// TwinCAT 3 PLC project BE_BUZ_Neutal
// ProgramVersion: 3.1.4023.0
// libraries:
//   EfficientIO Communicator, * (EfficientIO)
//   Lynus Persistent Data V1, * (Lynus AG)
//   Lynus Standards, * (Lynus AG)
//   Tc2_Standard, * (Beckhoff Automation GmbH)
//   Tc2_System, * (Beckhoff Automation GmbH)
//   Tc2_TcpIp, * (Beckhoff Automation GmbH)
//   Tc2_Utilities, * (Beckhoff Automation GmbH)
//   Tc3_IotBase, * (Beckhoff Automation GmbH)
//   Tc3_JsonXml, * (Beckhoff Automation GmbH)
//   Tc3_Module, * (Beckhoff Automation GmbH)
// project tree:
//   / FastTask.TcTTO, MiddleTask.TcTTO, SlowTask.TcTTO
//   FB/ fb_Convert4BytesToLreal.TcPOU, FB_OCHSNER_Web2Com1.TcPOU, FB_OCHSNER_Web2Com2.TcPOU, FB_OCHSNER_Web2Com2_Helper.TcPOU, FB_OCHSNER_Web2Com3_Helper.TcPOU, FB_OCHSNER_Web2Com3.TcPOU, FB_OCHSNER_Web2Com1_Helper.TcPOU, FB_OCHSNER_Web2Com4.TcPOU, FB_OCHSNER_Web2Com4_Helper.TcPOU, FB_TCPModbusRequest_Grid.TcPOU, FB_TCPModbusRequest_PV.TcPOU
//   POUs/ prgComEffIO.TcPOU, prgGrid.TcPOU, prgHP1.TcPOU, prgHP2.TcPOU, prgHP3.TcPOU, prgHP4.TcPOU, prgPersistent.TcPOU, prgPV.TcPOU, prgRWEffIO.TcPOU, prgVarEffIO.TcPOU
// real-time tasks:
//   TASK MiddleTask: cycle T#10ms, priority 8, ADS port 350
//   TASK FastTask: cycle T#5ms, priority 6, ADS port 351
//   TASK SlowTask: cycle T#20ms, priority 10, ADS port 352

CONFIGURATION BE_BUZ_Neutal
    RESOURCE PLC ON TwinCAT3
        TASK FastTask(INTERVAL := T#5ms, PRIORITY := 6);
        TASK MiddleTask(INTERVAL := T#10ms, PRIORITY := 8);
        TASK SlowTask(INTERVAL := T#20ms, PRIORITY := 10);
        PROGRAM prgRWEffIO WITH FastTask : prgRWEffIO;
        PROGRAM prgVarEffIO WITH FastTask : prgVarEffIO;
        PROGRAM prgHP1 WITH MiddleTask : prgHP1;
        PROGRAM prgHP3 WITH MiddleTask : prgHP3;
        PROGRAM prgHP2 WITH MiddleTask : prgHP2;
        PROGRAM prgHP4 WITH MiddleTask : prgHP4;
        PROGRAM prgPV WITH MiddleTask : prgPV;
        PROGRAM prgPersistent WITH MiddleTask : prgPersistent;
        PROGRAM prgComEffIO WITH SlowTask : prgComEffIO;
    END_RESOURCE
END_CONFIGURATION

// ---- POUs/prgRWEffIO.TcPOU
PROGRAM prgRWEffIO
VAR
	fbRW1		: FB_ReadWrite_V2;
END_VAR

fbRW1(
	eUploadType:= eSelectDataUploadType.e_Change_Intervall5min, 
	bBusy=> , 
	bError=> , 
	udiErrorCodeOut=> ,
	eErrorReadWrite_Out=> );

END_PROGRAM

// ---- POUs/prgVarEffIO.TcPOU
PROGRAM prgVarEffIO
VAR
	fbVar			: FB_VarInfo;
END_VAR

fbVar(
	bReadInfo:= , 
	eTMCFile:= eSelectTMCFile.eDontUseTMCFile, 
	eSavePositionTMCFile:= eSavePositionOnPLC.ePostionHardDisk, 
	udiCounterFoundVariables=> , 
	bError=> , 
	bBusy=> , 
	byProgress=> , 
	udiErrorCodeOut=> , 
	eErrorVarInfo_Out=> , 
	sVarWithError=> );

END_PROGRAM

// ---- POUs/prgHP1.TcPOU
PROGRAM prgHP1
VAR
	fbWb2Com1						: FB_OCHSNER_Web2Com1;
	byHP1StateHeatProd		: BYTE;		//{#lynus.ag#()}
	lrHP1TWVtemp			: LREAL;	//{#lynus.ag#()}
	lrHP1TWRtemp			: LREAL;	//{#lynus.ag#()}
	lrHP1TQAtemp			: LREAL;	//{#lynus.ag#()}
	lrHP1TQEtemp			: LREAL;	//{#lynus.ag#()}
	lrHP1ThEnergykWh		: LREAL;	//{#lynus.ag#()}
	lrHP1ThEnergyMWh		: LREAL;	//{#lynus.ag#()}
	byHC1StateHC			: BYTE;		//{#lynus.ag#()}
	lrHC1OutTemp			: LREAL;	//{#lynus.ag#()}
	lrHC1OutTempAvg			: LREAL;	//{#lynus.ag#()}
	lrHC1SPRoomTemp			: LREAL;	//{#lynus.ag#()}
	lrHC1PreFlowTemp		: LREAL;	//{#lynus.ag#()}
	lrHC1SPFlowTemp			: LREAL;	//{#lynus.ag#()}
	byHP2StateHeatProd		: BYTE;		//{#lynus.ag#()}
	lrHP2TWVtemp			: LREAL;	//{#lynus.ag#()}
	lrHP2TWRtemp			: LREAL;	//{#lynus.ag#()}
	lrHP2TQAtemp			: LREAL;	//{#lynus.ag#()}
	lrHP2TQEtemp			: LREAL;	//{#lynus.ag#()}
	lrHP2ThEnergykWh		: LREAL;	//{#lynus.ag#()}
	lrHP2ThEnergyMWh		: LREAL;	//{#lynus.ag#()}
END_VAR

fbWb2Com1(
	bStart:= TRUE, 
	tDelayRequest:= T#60S, 
	sHostname:= 'localhost', 
	bValidResult=> , 
	bBusy=> , 
	bError=> , 
	bDone=> , 
	hrErrorCode=> ,
	byHP1StateHeatProd => byHP1StateHeatProd,
	lrHP1TWVtemp => lrHP1TWVtemp,
	lrHP1TWRtemp => lrHP1TWRtemp,
	lrHP1TQAtemp => lrHP1TQAtemp,
	lrHP1TQEtemp => lrHP1TQEtemp,
	lrHP1ThEnergykWh => lrHP1ThEnergykWh,
	lrHP1ThEnergyMWh => lrHP1ThEnergyMWh,
	byHC1StateHC => byHC1StateHC,
	lrHC1OutTemp => lrHC1OutTemp,
	lrHC1OutTempAvg => lrHC1OutTempAvg,
	lrHC1SPRoomTemp => lrHC1SPRoomTemp,
	lrHC1PreFlowTemp => lrHC1PreFlowTemp,
	lrHC1SPFlowTemp => lrHC1SPFlowTemp,
	byHP2StateHeatProd => byHP2StateHeatProd,
	lrHP2TWVtemp => lrHP2TWVtemp,
	lrHP2TWRtemp => lrHP2TWRtemp,
	lrHP2TQAtemp => lrHP2TQAtemp,
	lrHP2TQEtemp => lrHP2TQEtemp,
	lrHP2ThEnergykWh => lrHP2ThEnergykWh,
	lrHP2ThEnergyMWh => lrHP2ThEnergyMWh);

END_PROGRAM

// ---- FB/FB_OCHSNER_Web2Com1.TcPOU
FUNCTION_BLOCK FB_OCHSNER_Web2Com1
VAR_INPUT
	bStart				: BOOL;
	tDelayRequest		: TIME;		//Timer for delay before start with the next read or write Request
	sHostname			: STRING(255);		//Hostname or IP Adress from the Server
END_VAR

VAR_IN_OUT
END_VAR

VAR_OUTPUT
	bValidResult		: BOOL;							//Valid Result received from Server
    bBusy				: BOOL;							//Function is Busy
    bError				: BOOL;							//Error sucess
	bDone				: BOOL;							//True after the decoding from the received Json File
	bConnected			: BOOL;							//Connection to the Server
	hrErrorCode       	: HRESULT;						//Error Result from Http Client
	byHP1StateHeatProd		: BYTE;
	lrHP1TWVtemp			: LREAL;
	lrHP1TWRtemp			: LREAL;
	lrHP1TQAtemp			: LREAL;
	lrHP1TQEtemp			: LREAL;
	lrHP1ThEnergykWh		: LREAL;
	lrHP1ThEnergyMWh		: LREAL;
	byHC1StateHC			: BYTE;
	lrHC1OutTemp			: LREAL;
	lrHC1OutTempAvg			: LREAL;
	lrHC1SPRoomTemp			: LREAL;
	lrHC1PreFlowTemp		: LREAL;
	lrHC1SPFlowTemp			: LREAL;
	byHP2StateHeatProd		: BYTE;
	lrHP2TWVtemp			: LREAL;
	lrHP2TWRtemp			: LREAL;
	lrHP2TQAtemp			: LREAL;
	lrHP2TQEtemp			: LREAL;
	lrHP2ThEnergykWh		: LREAL;
	lrHP2ThEnergyMWh		: LREAL;
END_VAR

VAR
	fbClient			: FB_IotHttpClient;
	fbHttpGet			: FB_OCHSNER_Web2Com1_Helper;
	timStartRequest		: TON;							//Timer to Start the Request
	FPStartRequest		: R_TRIG;						//Internal positive Edge
	FPDone				: R_TRIG;						//Internal positive Edge
	FNStart				: F_TRIG;						//Internal negative Edge
END_VAR

(*------------------------------------------------------------------------------------Configure HTTP Client------------------------------------------------------------------------------------------------------*)

fbClient.sHostName := sHostname;
fbClient.tConnectionTimeout := T#20S;
fbClient.bKeepAlive := FALSE;

IF NOT fbClient.bConfigured THEN 
	fbClient.nHostPort:= 80;
	fbClient.bKeepAlive := FALSE;
	fbClient.tConnectionTimeout := T#20S;
END_IF


//Timer to start the Request
FPStartRequest(CLK:= bStart, Q=> );
	timStartRequest(IN:= fbClient.bConfigured AND bStart AND NOT timStartRequest.Q, PT:= tDelayRequest, Q=> , ET=> );
		IF ((timStartRequest.Q AND NOT bBusy) OR (FPStartRequest.Q AND NOT bBusy AND fbClient.bConfigured)) THEN fbHttpGet.bSend := TRUE; END_IF

				
//Http Get Function
fbHttpGet(
	bSend:= , 
	fbClient:= fbClient, 
	bBusy=> bBusy, 
	bError=> ,
	byHP1StateHeatProd => byHP1StateHeatProd,
	lrHP1TWVtemp => lrHP1TWVtemp,
	lrHP1TWRtemp => lrHP1TWRtemp,
	lrHP1TQAtemp => lrHP1TQAtemp,
	lrHP1TQEtemp => lrHP1TQEtemp,
	lrHP1ThEnergykWh => lrHP1ThEnergykWh,
	lrHP1ThEnergyMWh => lrHP1ThEnergyMWh,
	byHC1StateHC => byHC1StateHC,
	lrHC1OutTemp => lrHC1OutTemp,
	lrHC1OutTempAvg => lrHC1OutTempAvg,
	lrHC1SPRoomTemp => lrHC1SPRoomTemp,
	lrHC1PreFlowTemp => lrHC1PreFlowTemp,
	lrHC1SPFlowTemp => lrHC1SPFlowTemp,
	byHP2StateHeatProd => byHP2StateHeatProd,
	lrHP2TWVtemp => lrHP2TWVtemp,
	lrHP2TWRtemp => lrHP2TWRtemp,
	lrHP2TQAtemp => lrHP2TQAtemp,
	lrHP2TQEtemp => lrHP2TQEtemp,
	lrHP2ThEnergykWh => lrHP2ThEnergykWh,
	lrHP2ThEnergyMWh => lrHP2ThEnergyMWh );


fbHttpGet.bSend := FALSE;

FPDone(CLK:= bDone, Q=> );

fbClient.Execute();

//Error
IF fbHttpGet.bError OR fbClient.bError THEN bError := TRUE; ELSE bError := FALSE; END_IF	
	hrErrorCode := fbClient.hrErrorCode;

END_FUNCTION_BLOCK

// ---- FB/FB_OCHSNER_Web2Com1_Helper.TcPOU
FUNCTION_BLOCK FB_OCHSNER_Web2Com1_Helper
VAR_INPUT
	bSend				: BOOL;
END_VAR

VAR_IN_OUT
	fbClient			: FB_IotHttpClient;
END_VAR

VAR_OUTPUT
	bBusy				: BOOL;
	bError				: BOOL;
	byHP1StateHeatProd		: BYTE;
	lrHP1TWVtemp			: LREAL;
	lrHP1TWRtemp			: LREAL;
	lrHP1TQAtemp			: LREAL;
	lrHP1TQEtemp			: LREAL;
	lrHP1ThEnergykWh		: LREAL;
	lrHP1ThEnergyMWh		: LREAL;
	byHC1StateHC			: BYTE;
	lrHC1OutTemp			: LREAL;
	lrHC1OutTempAvg			: LREAL;
	lrHC1SPRoomTemp			: LREAL;
	lrHC1PreFlowTemp		: LREAL;
	lrHC1SPFlowTemp			: LREAL;
	byHP2StateHeatProd		: BYTE;
	lrHP2TWVtemp			: LREAL;
	lrHP2TWRtemp			: LREAL;
	lrHP2TQAtemp			: LREAL;
	lrHP2TQEtemp			: LREAL;
	lrHP2ThEnergykWh		: LREAL;
	lrHP2ThEnergyMWh		: LREAL;
END_VAR

VAR
	fbRequest1			: FB_IotHttpRequest;
	fbRequest2			: FB_IotHttpRequest;
	fbRequest3			: FB_IotHttpRequest;

	fbJson				: FB_JsonDomParser;
	nState				: UDINT;
	RisingEdge			: R_TRIG;
	timTimeout			: TON;
	tTimeOut			: TIME := T#90S;
	bGetContentResult	: BOOL;
	sContent1			: STRING(511);
	sContent2			: STRING(511);
	sContent3			: STRING(511);
	
	bGetJsonResult		: BOOL;
	jsonDoc				: SJsonValue;
	jsonVal				: SJsonValue;
	
	nReqCount			: UDINT;	
	nResCount			: UDINT;
	nValidResCount		: UDINT;
	nErrCount			: UDINT;
END_VAR

//Timer for Timeout
timTimeout(IN:= nState = 1 AND bBusy, PT:= tTimeOut, Q=> , ET=> );
	IF timTimeout.Q THEN 
		nState := 0;
		bBusy := FALSE;
	END_IF

RisingEdge(CLK:= bSend );
CASE nState OF
0:	
	IF RisingEdge.Q THEN 
		IF 
			fbRequest1.SendRequest(sUri:='/web2com_1HP1.php', fbClient:=fbClient, eRequestType:=ETcIotHttpRequestType.HTTP_Get, 0, 0, 0) AND
			fbRequest2.SendRequest(sUri:='/web2com_1HC1.php', fbClient:=fbClient, eRequestType:=ETcIotHttpRequestType.HTTP_Get, 0, 0, 0) AND 
			fbRequest3.SendRequest(sUri:='/web2com_1HP2.php', fbClient:=fbClient, eRequestType:=ETcIotHttpRequestType.HTTP_Get, 0, 0, 0) THEN				
			nState:= 1;
			nReqCount:= nReqCount+1;
			bBusy:= TRUE;
			bError:= FALSE;
		END_IF					
	END_IF
1:
	IF NOT fbRequest1.bBusy AND NOT fbRequest2.bBusy AND NOT fbRequest3.bBusy THEN
		bError:= TRUE;
		IF NOT fbRequest1.bError THEN				 
			bGetContentResult:= fbRequest1.GetContent(pContent:= ADR(sContent1), nContentSize:= SIZEOF(sContent1), bSetNullTermination:= TRUE);
			IF fbRequest1.nStatusCode >= 200 AND fbRequest1.nStatusCode < 300 THEN
				bGetJsonResult:= FALSE;
				jsonDoc:= fbRequest1.GetJsonDomContent(fbJson);
				IF jsonDoc <> 0 THEN
					bGetJsonResult:= TRUE;
					IF fbJson.HasMember(jsonDoc, '1211250')  THEN
						jsonVal:= fbJson.FindMember(jsonDoc, '1211250');
						nValidResCount:= nValidResCount+1;
						IF fbJson.IsNumber(jsonVal) THEN							
							byHP1StateHeatProd := DINT_TO_BYTE(fbJson.GetInt(jsonVal));									
						END_IF
						
						jsonVal:= fbJson.FindMember(jsonDoc, '1211251');
						nValidResCount:= nValidResCount+1;
						IF fbJson.IsDouble(jsonVal) THEN							
							lrHP1TWVtemp := fbJson.GetDouble(jsonVal);									
						END_IF
						
						jsonVal:= fbJson.FindMember(jsonDoc, '1211253');
						nValidResCount:= nValidResCount+1;
						IF fbJson.IsDouble(jsonVal) THEN							
							lrHP1TWRtemp := fbJson.GetDouble(jsonVal);									
						END_IF
						
						jsonVal:= fbJson.FindMember(jsonDoc, '1211254');
						nValidResCount:= nValidResCount+1;
						IF fbJson.IsDouble(jsonVal) THEN							
							lrHP1TQAtemp := fbJson.GetDouble(jsonVal);									
						END_IF
						
						jsonVal:= fbJson.FindMember(jsonDoc, '1211255');
						nValidResCount:= nValidResCount+1;
						IF fbJson.IsDouble(jsonVal) THEN							
							lrHP1TQEtemp := fbJson.GetDouble(jsonVal);									
						END_IF
						
						jsonVal:= fbJson.FindMember(jsonDoc, '1211258');
						nValidResCount:= nValidResCount+1;
						IF fbJson.IsNumber(jsonVal) THEN							
							lrHP1ThEnergykWh := fbJson.GetDouble(jsonVal);									
						END_IF
						
						jsonVal:= fbJson.FindMember(jsonDoc, '1211259');
						nValidResCount:= nValidResCount+1;
						IF fbJson.IsNumber(jsonVal) THEN							
							lrHP1ThEnergyMWh := fbJson.GetDouble(jsonVal);									
						END_IF
						
						bError:= FALSE;
						END_IF
					END_IF						
				nResCount:= nResCount+1;			
				END_IF
		END_IF
		
		IF NOT fbRequest2.bError THEN				 
			bGetContentResult:= fbRequest2.GetContent(pContent:= ADR(sContent2), nContentSize:= SIZEOF(sContent2), bSetNullTermination:= TRUE);
			IF fbRequest2.nStatusCode >= 200 AND fbRequest2.nStatusCode < 300 THEN
				bGetJsonResult:= FALSE;
				jsonDoc:= fbRequest2.GetJsonDomContent(fbJson);
				IF jsonDoc <> 0 THEN
					bGetJsonResult:= TRUE;
					IF fbJson.HasMember(jsonDoc, '1241190')  THEN
						jsonVal:= fbJson.FindMember(jsonDoc, '1241190');
						nValidResCount:= nValidResCount+1;
						IF fbJson.IsNumber(jsonVal) THEN							
							byHC1StateHC := DINT_TO_BYTE(fbJson.GetInt(jsonVal));									
						END_IF
						
						jsonVal:= fbJson.FindMember(jsonDoc, '1241191');
						nValidResCount:= nValidResCount+1;
						IF fbJson.IsDouble(jsonVal) THEN							
							lrHC1OutTemp := fbJson.GetDouble(jsonVal);									
						END_IF
						
						jsonVal:= fbJson.FindMember(jsonDoc, '1241192');
						nValidResCount:= nValidResCount+1;
						IF fbJson.IsDouble(jsonVal) THEN							
							lrHC1OutTempAvg := fbJson.GetDouble(jsonVal);									
						END_IF
						
						jsonVal:= fbJson.FindMember(jsonDoc, '1241193');
						nValidResCount:= nValidResCount+1;
						IF fbJson.IsDouble(jsonVal) THEN							
							lrHC1SPRoomTemp := fbJson.GetDouble(jsonVal);									
						END_IF
						
						jsonVal:= fbJson.FindMember(jsonDoc, '1241194');
						nValidResCount:= nValidResCount+1;
						IF fbJson.IsDouble(jsonVal) THEN							
							lrHC1PreFlowTemp := fbJson.GetDouble(jsonVal);									
						END_IF
						
						jsonVal:= fbJson.FindMember(jsonDoc, '1241195');
						nValidResCount:= nValidResCount+1;
						IF fbJson.IsDouble(jsonVal) THEN							
							lrHC1SPFlowTemp := fbJson.GetDouble(jsonVal);									
						END_IF
						
						bError:= FALSE;
						END_IF
					END_IF						
				nResCount:= nResCount+1;			
				END_IF
		END_IF
		
		IF NOT fbRequest3.bError THEN				 
			bGetContentResult:= fbRequest3.GetContent(pContent:= ADR(sContent3), nContentSize:= SIZEOF(sContent3), bSetNullTermination:= TRUE);
			IF fbRequest3.nStatusCode >= 200 AND fbRequest3.nStatusCode < 300 THEN
				bGetJsonResult:= FALSE;
				jsonDoc:= fbRequest3.GetJsonDomContent(fbJson);
				IF jsonDoc <> 0 THEN
					bGetJsonResult:= TRUE;
					IF fbJson.HasMember(jsonDoc, '1311250')  THEN
						jsonVal:= fbJson.FindMember(jsonDoc, '1311250');
						nValidResCount:= nValidResCount+1;
						IF fbJson.IsNumber(jsonVal) THEN							
							byHP2StateHeatProd := DINT_TO_BYTE(fbJson.GetInt(jsonVal));									
						END_IF
						
						jsonVal:= fbJson.FindMember(jsonDoc, '1311251');
						nValidResCount:= nValidResCount+1;
						IF fbJson.IsDouble(jsonVal) THEN							
							lrHP2TWVtemp := fbJson.GetDouble(jsonVal);									
						END_IF
						
						jsonVal:= fbJson.FindMember(jsonDoc, '1311253');
						nValidResCount:= nValidResCount+1;
						IF fbJson.IsDouble(jsonVal) THEN							
							lrHP2TWRtemp := fbJson.GetDouble(jsonVal);									
						END_IF
						
						jsonVal:= fbJson.FindMember(jsonDoc, '1311254');
						nValidResCount:= nValidResCount+1;
						IF fbJson.IsDouble(jsonVal) THEN							
							lrHP2TQAtemp := fbJson.GetDouble(jsonVal);									
						END_IF
						
						jsonVal:= fbJson.FindMember(jsonDoc, '1311255');
						nValidResCount:= nValidResCount+1;
						IF fbJson.IsDouble(jsonVal) THEN							
							lrHP2TQEtemp := fbJson.GetDouble(jsonVal);									
						END_IF
						
						jsonVal:= fbJson.FindMember(jsonDoc, '1311258');
						nValidResCount:= nValidResCount+1;
						IF fbJson.IsNumber(jsonVal) THEN							
							lrHP2ThEnergykWh := fbJson.GetDouble(jsonVal);									
						END_IF
						
						jsonVal:= fbJson.FindMember(jsonDoc, '1311259');
						nValidResCount:= nValidResCount+1;
						IF fbJson.IsNumber(jsonVal) THEN							
							lrHP2ThEnergyMWh := fbJson.GetDouble(jsonVal);									
						END_IF
						
						bError:= FALSE;
						END_IF
					END_IF						
				nResCount:= nResCount+1;			
				END_IF
		END_IF
		
		nState:= 0;
		bBusy:= FALSE;
		IF bError THEN
			nErrCount:= nErrCount+1;
		END_IF
	END_IF  	
END_CASE

END_FUNCTION_BLOCK

// ---- POUs/prgHP3.TcPOU
PROGRAM prgHP3
VAR
	fbWb2Com3						: FB_OCHSNER_Web2Com3;
	byHP1StateHeatProd		: BYTE;		//{#lynus.ag#()}
	lrHP1TWVtemp			: LREAL;	//{#lynus.ag#()}
	lrHP1TWRtemp			: LREAL;	//{#lynus.ag#()}
	lrHP1TQAtemp			: LREAL;	//{#lynus.ag#()}
	lrHP1TQEtemp			: LREAL;	//{#lynus.ag#()}
	lrHP1ThEnergykWh		: LREAL;	//{#lynus.ag#()}
	lrHP1ThEnergyMWh		: LREAL;	//{#lynus.ag#()}
	byHC1StateHC			: BYTE;		//{#lynus.ag#()}
	lrHC1OutTemp			: LREAL;	//{#lynus.ag#()}
	lrHC1OutTempAvg			: LREAL;	//{#lynus.ag#()}
	lrHC1RoomTemp			: LREAL;	//{#lynus.ag#()}
	lrHC1SPRoomTemp			: LREAL;	//{#lynus.ag#()}
	lrHC1PreFlowTemp		: LREAL;	//{#lynus.ag#()}
	lrHC1SPFlowTemp			: LREAL;	//{#lynus.ag#()}
END_VAR

fbWb2Com3(
	bStart:= TRUE, 
	tDelayRequest:= T#60S, 
	sHostname:= 'localhost', 
	bValidResult=> , 
	bBusy=> , 
	bError=> , 
	bDone=> , 
	hrErrorCode=> ,
	byHP1StateHeatProd => byHP1StateHeatProd,
	lrHP1TWVtemp => lrHP1TWVtemp,
	lrHP1TWRtemp => lrHP1TWRtemp,
	lrHP1TQAtemp => lrHP1TQAtemp,
	lrHP1TQEtemp => lrHP1TQEtemp,
	lrHP1ThEnergykWh => lrHP1ThEnergykWh,
	lrHP1ThEnergyMWh => lrHP1ThEnergyMWh,
	byHC1StateHC => byHC1StateHC,
	lrHC1OutTemp => lrHC1OutTemp,
	lrHC1OutTempAvg => lrHC1OutTempAvg,
	lrHC1RoomTemp => lrHC1RoomTemp,
	lrHC1SPRoomTemp => lrHC1SPRoomTemp,
	lrHC1PreFlowTemp => lrHC1PreFlowTemp,
	lrHC1SPFlowTemp => lrHC1SPFlowTemp);

END_PROGRAM

// ---- FB/FB_OCHSNER_Web2Com3.TcPOU
FUNCTION_BLOCK FB_OCHSNER_Web2Com3
VAR_INPUT
	bStart				: BOOL;
	tDelayRequest		: TIME;		//Timer for delay before start with the next read or write Request
	sHostname			: STRING(255);		//Hostname or IP Adress from the Server
END_VAR

VAR_IN_OUT
END_VAR

VAR_OUTPUT
	bValidResult		: BOOL;							//Valid Result received from Server
    bBusy				: BOOL;							//Function is Busy
    bError				: BOOL;							//Error sucess
	bDone				: BOOL;							//True after the decoding from the received Json File
	bConnected			: BOOL;							//Connection to the Server
	hrErrorCode       	: HRESULT;						//Error Result from Http Client
	byHP1StateHeatProd		: BYTE;
	lrHP1TWVtemp			: LREAL;
	lrHP1TWRtemp			: LREAL;
	lrHP1TQAtemp			: LREAL;
	lrHP1TQEtemp			: LREAL;
	lrHP1ThEnergykWh		: LREAL;
	lrHP1ThEnergyMWh		: LREAL;
	byHC1StateHC			: BYTE;
	lrHC1OutTemp			: LREAL;
	lrHC1OutTempAvg			: LREAL;
	lrHC1RoomTemp			: LREAL;
	lrHC1SPRoomTemp			: LREAL;
	lrHC1PreFlowTemp		: LREAL;
	lrHC1SPFlowTemp			: LREAL;
END_VAR

VAR
	fbClient			: FB_IotHttpClient;
	fbHttpGet			: FB_OCHSNER_Web2Com3_Helper;
	timStartRequest		: TON;							//Timer to Start the Request
	FPStartRequest		: R_TRIG;						//Internal positive Edge
	FPDone				: R_TRIG;						//Internal positive Edge
	FNStart				: F_TRIG;						//Internal negative Edge
END_VAR

(*------------------------------------------------------------------------------------Configure HTTP Client------------------------------------------------------------------------------------------------------*)

fbClient.sHostName := sHostname;
fbClient.tConnectionTimeout := T#20S;
fbClient.bKeepAlive := FALSE;

IF NOT fbClient.bConfigured THEN 
	fbClient.nHostPort:= 80;
	fbClient.bKeepAlive := FALSE;
	fbClient.tConnectionTimeout := T#20S;
END_IF


//Timer to start the Request
FPStartRequest(CLK:= bStart, Q=> );
	timStartRequest(IN:= fbClient.bConfigured AND bStart AND NOT timStartRequest.Q, PT:= tDelayRequest, Q=> , ET=> );
		IF ((timStartRequest.Q AND NOT bBusy) OR (FPStartRequest.Q AND NOT bBusy AND fbClient.bConfigured)) THEN fbHttpGet.bSend := TRUE; END_IF

				
//Http Get Function
fbHttpGet(
	bSend:= , 
	fbClient:= fbClient, 
	bBusy=> bBusy, 
	bError=> ,
	byHP1StateHeatProd => byHP1StateHeatProd,
	lrHP1TWVtemp => lrHP1TWVtemp,
	lrHP1TWRtemp => lrHP1TWRtemp,
	lrHP1TQAtemp => lrHP1TQAtemp,
	lrHP1TQEtemp => lrHP1TQEtemp,
	lrHP1ThEnergykWh => lrHP1ThEnergykWh,
	lrHP1ThEnergyMWh => lrHP1ThEnergyMWh,
	byHC1StateHC => byHC1StateHC,
	lrHC1OutTemp => lrHC1OutTemp,
	lrHC1OutTempAvg => lrHC1OutTempAvg,
	lrHC1RoomTemp => lrHC1RoomTemp,
	lrHC1SPRoomTemp => lrHC1SPRoomTemp,
	lrHC1PreFlowTemp => lrHC1PreFlowTemp,
	lrHC1SPFlowTemp => lrHC1SPFlowTemp);


fbHttpGet.bSend := FALSE;

FPDone(CLK:= bDone, Q=> );

fbClient.Execute();

//Error
IF fbHttpGet.bError OR fbClient.bError THEN bError := TRUE; ELSE bError := FALSE; END_IF	
	hrErrorCode := fbClient.hrErrorCode;

END_FUNCTION_BLOCK

// ---- FB/FB_OCHSNER_Web2Com3_Helper.TcPOU
FUNCTION_BLOCK FB_OCHSNER_Web2Com3_Helper
VAR_INPUT
	bSend				: BOOL;
END_VAR

VAR_IN_OUT
	fbClient			: FB_IotHttpClient;
END_VAR

VAR_OUTPUT
	bBusy				: BOOL;
	bError				: BOOL;
	byHP1StateHeatProd		: BYTE;
	lrHP1TWVtemp			: LREAL;
	lrHP1TWRtemp			: LREAL;
	lrHP1TQAtemp			: LREAL;
	lrHP1TQEtemp			: LREAL;
	lrHP1ThEnergykWh		: LREAL;
	lrHP1ThEnergyMWh		: LREAL;
	byHC1StateHC			: BYTE;
	lrHC1OutTemp			: LREAL;
	lrHC1OutTempAvg			: LREAL;
	lrHC1RoomTemp			: LREAL;
	lrHC1SPRoomTemp			: LREAL;
	lrHC1PreFlowTemp		: LREAL;
	lrHC1SPFlowTemp			: LREAL;
END_VAR

VAR
	fbRequest1			: FB_IotHttpRequest;
	fbRequest2			: FB_IotHttpRequest;

	fbJson				: FB_JsonDomParser;
	nState				: UDINT;
	RisingEdge			: R_TRIG;
	timTimeout			: TON;
	tTimeOut			: TIME := T#90S;
	bGetContentResult	: BOOL;
	sContent1			: STRING(511);
	sContent2			: STRING(511);
	
	bGetJsonResult		: BOOL;
	jsonDoc				: SJsonValue;
	jsonVal				: SJsonValue;
	
	nReqCount			: UDINT;	
	nResCount			: UDINT;
	nValidResCount		: UDINT;
	nErrCount			: UDINT;
END_VAR

//Timer for Timeout
timTimeout(IN:= nState = 1 AND bBusy, PT:= tTimeOut, Q=> , ET=> );
	IF timTimeout.Q THEN 
		nState := 0;
		bBusy := FALSE;
	END_IF

RisingEdge(CLK:= bSend );
CASE nState OF
0:	
	IF RisingEdge.Q THEN 
		IF 
			fbRequest1.SendRequest(sUri:='/web2com_3HP1.php', fbClient:=fbClient, eRequestType:=ETcIotHttpRequestType.HTTP_Get, 0, 0, 0) AND
			fbRequest2.SendRequest(sUri:='/web2com_3HC1.php', fbClient:=fbClient, eRequestType:=ETcIotHttpRequestType.HTTP_Get, 0, 0, 0) THEN				
			nState:= 1;
			nReqCount:= nReqCount+1;
			bBusy:= TRUE;
			bError:= FALSE;
		END_IF					
	END_IF
1:
	IF NOT fbRequest1.bBusy AND NOT fbRequest2.bBusy THEN
		bError:= TRUE;
		IF NOT fbRequest1.bError THEN				 
			bGetContentResult:= fbRequest1.GetContent(pContent:= ADR(sContent1), nContentSize:= SIZEOF(sContent1), bSetNullTermination:= TRUE);
			IF fbRequest1.nStatusCode >= 200 AND fbRequest1.nStatusCode < 300 THEN
				bGetJsonResult:= FALSE;
				jsonDoc:= fbRequest1.GetJsonDomContent(fbJson);
				IF jsonDoc <> 0 THEN
					bGetJsonResult:= TRUE;
					IF fbJson.HasMember(jsonDoc, '1211250')  THEN
						jsonVal:= fbJson.FindMember(jsonDoc, '1211250');
						nValidResCount:= nValidResCount+1;
						IF fbJson.IsNumber(jsonVal) THEN							
							byHP1StateHeatProd := DINT_TO_BYTE(fbJson.GetInt(jsonVal));									
						END_IF
						
						jsonVal:= fbJson.FindMember(jsonDoc, '1211251');
						nValidResCount:= nValidResCount+1;
						IF fbJson.IsDouble(jsonVal) THEN							
							lrHP1TWVtemp := fbJson.GetDouble(jsonVal);									
						END_IF
						
						jsonVal:= fbJson.FindMember(jsonDoc, '1211253');
						nValidResCount:= nValidResCount+1;
						IF fbJson.IsDouble(jsonVal) THEN							
							lrHP1TWRtemp := fbJson.GetDouble(jsonVal);									
						END_IF
						
						jsonVal:= fbJson.FindMember(jsonDoc, '1211254');
						nValidResCount:= nValidResCount+1;
						IF fbJson.IsDouble(jsonVal) THEN							
							lrHP1TQAtemp := fbJson.GetDouble(jsonVal);									
						END_IF
						
						jsonVal:= fbJson.FindMember(jsonDoc, '1211255');
						nValidResCount:= nValidResCount+1;
						IF fbJson.IsDouble(jsonVal) THEN							
							lrHP1TQEtemp := fbJson.GetDouble(jsonVal);									
						END_IF
						
						jsonVal:= fbJson.FindMember(jsonDoc, '1211258');
						nValidResCount:= nValidResCount+1;
						IF fbJson.IsNumber(jsonVal) THEN							
							lrHP1ThEnergykWh := fbJson.GetDouble(jsonVal);									
						END_IF
						
						jsonVal:= fbJson.FindMember(jsonDoc, '1211259');
						nValidResCount:= nValidResCount+1;
						IF fbJson.IsNumber(jsonVal) THEN							
							lrHP1ThEnergyMWh := fbJson.GetDouble(jsonVal);									
						END_IF
						
						bError:= FALSE;
						END_IF
					END_IF						
				nResCount:= nResCount+1;			
				END_IF
		END_IF
		
		IF NOT fbRequest2.bError THEN				 
			bGetContentResult:= fbRequest2.GetContent(pContent:= ADR(sContent2), nContentSize:= SIZEOF(sContent2), bSetNullTermination:= TRUE);
			IF fbRequest2.nStatusCode >= 200 AND fbRequest2.nStatusCode < 300 THEN
				bGetJsonResult:= FALSE;
				jsonDoc:= fbRequest2.GetJsonDomContent(fbJson);
				IF jsonDoc <> 0 THEN
					bGetJsonResult:= TRUE;
					IF fbJson.HasMember(jsonDoc, '1241190')  THEN
						jsonVal:= fbJson.FindMember(jsonDoc, '1241190');
						nValidResCount:= nValidResCount+1;
						IF fbJson.IsNumber(jsonVal) THEN							
							byHC1StateHC := DINT_TO_BYTE(fbJson.GetInt(jsonVal));									
						END_IF
						
						jsonVal:= fbJson.FindMember(jsonDoc, '1241191');
						nValidResCount:= nValidResCount+1;
						IF fbJson.IsDouble(jsonVal) THEN							
							lrHC1OutTemp := fbJson.GetDouble(jsonVal);									
						END_IF
						
						jsonVal:= fbJson.FindMember(jsonDoc, '1241192');
						nValidResCount:= nValidResCount+1;
						IF fbJson.IsDouble(jsonVal) THEN							
							lrHC1OutTempAvg := fbJson.GetDouble(jsonVal);									
						END_IF
						
						jsonVal:= fbJson.FindMember(jsonDoc, '1241193');
						nValidResCount:= nValidResCount+1;
						IF fbJson.IsDouble(jsonVal) THEN							
							lrHC1RoomTemp := fbJson.GetDouble(jsonVal);									
						END_IF
						
						jsonVal:= fbJson.FindMember(jsonDoc, '1241194');
						nValidResCount:= nValidResCount+1;
						IF fbJson.IsDouble(jsonVal) THEN							
							lrHC1SPRoomTemp := fbJson.GetDouble(jsonVal);									
						END_IF
						
						jsonVal:= fbJson.FindMember(jsonDoc, '1241195');
						nValidResCount:= nValidResCount+1;
						IF fbJson.IsDouble(jsonVal) THEN							
							lrHC1PreFlowTemp := fbJson.GetDouble(jsonVal);									
						END_IF
						
						jsonVal:= fbJson.FindMember(jsonDoc, '1241196');
						nValidResCount:= nValidResCount+1;
						IF fbJson.IsDouble(jsonVal) THEN							
							lrHC1SPFlowTemp := fbJson.GetDouble(jsonVal);									
						END_IF
						
						bError:= FALSE;
						END_IF
					END_IF						
				nResCount:= nResCount+1;			
				END_IF
		END_IF
		
		nState:= 0;
		bBusy:= FALSE;
		IF bError THEN
			nErrCount:= nErrCount+1;
		END_IF
	END_IF  	
END_CASE

END_FUNCTION_BLOCK

// ---- POUs/prgHP2.TcPOU
PROGRAM prgHP2
VAR
	fbWb2Com2						: FB_OCHSNER_Web2Com2;
	byHP1StateHeatProd		: BYTE;		//{#lynus.ag#()}
	lrHP1TWVtemp			: LREAL;	//{#lynus.ag#()}
	lrHP1TWRtemp			: LREAL;	//{#lynus.ag#()}
	lrHP1TQAtemp			: LREAL;	//{#lynus.ag#()}
	lrHP1TQEtemp			: LREAL;	//{#lynus.ag#()}
	lrHP1ThEnergykWh		: LREAL;	//{#lynus.ag#()}
	lrHP1ThEnergyMWh		: LREAL;	//{#lynus.ag#()}
	byHC1StateHC			: BYTE;
	lrHC1OutTemp			: LREAL;
	lrHC1OutTempAvg			: LREAL;
	lrHC1SPRoomTemp			: LREAL;
	lrHC1PreFlowTemp		: LREAL;
	lrHC1SPFlowTemp			: LREAL;
END_VAR

fbWb2Com2(
	bStart:= TRUE, 
	tDelayRequest:= T#60S, 
	sHostname:= 'localhost', 
	bValidResult=> , 
	bBusy=> , 
	bError=> , 
	bDone=> , 
	hrErrorCode=> ,
	byHP1StateHeatProd => byHP1StateHeatProd,
	lrHP1TWVtemp => lrHP1TWVtemp,
	lrHP1TWRtemp => lrHP1TWRtemp,
	lrHP1TQAtemp => lrHP1TQAtemp,
	lrHP1TQEtemp => lrHP1TQEtemp,
	lrHP1ThEnergykWh => lrHP1ThEnergykWh,
	lrHP1ThEnergyMWh => lrHP1ThEnergyMWh,
	byHC1StateHC => byHC1StateHC,
	lrHC1OutTemp => lrHC1OutTemp,
	lrHC1OutTempAvg => lrHC1OutTempAvg,
	lrHC1SPRoomTemp => lrHC1SPRoomTemp,
	lrHC1PreFlowTemp => lrHC1PreFlowTemp,
	lrHC1SPFlowTemp => lrHC1SPFlowTemp);

END_PROGRAM

// ---- FB/FB_OCHSNER_Web2Com2.TcPOU
FUNCTION_BLOCK FB_OCHSNER_Web2Com2
VAR_INPUT
	bStart				: BOOL;
	tDelayRequest		: TIME;		//Timer for delay before start with the next read or write Request
	sHostname			: STRING(255);		//Hostname or IP Adress from the Server
END_VAR

VAR_IN_OUT
END_VAR

VAR_OUTPUT
	bValidResult		: BOOL;							//Valid Result received from Server
    bBusy				: BOOL;							//Function is Busy
    bError				: BOOL;							//Error sucess
	bDone				: BOOL;							//True after the decoding from the received Json File
	bConnected			: BOOL;							//Connection to the Server
	hrErrorCode       	: HRESULT;						//Error Result from Http Client
	byHP1StateHeatProd		: BYTE;
	lrHP1TWVtemp			: LREAL;
	lrHP1TWRtemp			: LREAL;
	lrHP1TQAtemp			: LREAL;
	lrHP1TQEtemp			: LREAL;
	lrHP1ThEnergykWh		: LREAL;
	lrHP1ThEnergyMWh		: LREAL;
	byHC1StateHC			: BYTE;
	lrHC1OutTemp			: LREAL;
	lrHC1OutTempAvg			: LREAL;
	lrHC1RoomTemp			: LREAL;
	lrHC1SPRoomTemp			: LREAL;
	lrHC1PreFlowTemp		: LREAL;
	lrHC1SPFlowTemp			: LREAL;
END_VAR

VAR
	fbClient			: FB_IotHttpClient;
	fbHttpGet			: FB_OCHSNER_Web2Com2_Helper;
	timStartRequest		: TON;							//Timer to Start the Request
	FPStartRequest		: R_TRIG;						//Internal positive Edge
	FPDone				: R_TRIG;						//Internal positive Edge
	FNStart				: F_TRIG;						//Internal negative Edge
END_VAR

(*------------------------------------------------------------------------------------Configure HTTP Client------------------------------------------------------------------------------------------------------*)

fbClient.sHostName := sHostname;
fbClient.tConnectionTimeout := T#20S;
fbClient.bKeepAlive := FALSE;

IF NOT fbClient.bConfigured THEN 
	fbClient.nHostPort:= 80;
	fbClient.bKeepAlive := FALSE;
	fbClient.tConnectionTimeout := T#20S;
END_IF


//Timer to start the Request
FPStartRequest(CLK:= bStart, Q=> );
	timStartRequest(IN:= fbClient.bConfigured AND bStart AND NOT timStartRequest.Q, PT:= tDelayRequest, Q=> , ET=> );
		IF ((timStartRequest.Q AND NOT bBusy) OR (FPStartRequest.Q AND NOT bBusy AND fbClient.bConfigured)) THEN fbHttpGet.bSend := TRUE; END_IF

				
//Http Get Function
fbHttpGet(
	bSend:= , 
	fbClient:= fbClient, 
	bBusy=> bBusy, 
	bError=> ,
	byHP1StateHeatProd => byHP1StateHeatProd,
	lrHP1TWVtemp => lrHP1TWVtemp,
	lrHP1TWRtemp => lrHP1TWRtemp,
	lrHP1TQAtemp => lrHP1TQAtemp,
	lrHP1TQEtemp => lrHP1TQEtemp,
	lrHP1ThEnergykWh => lrHP1ThEnergykWh,
	lrHP1ThEnergyMWh => lrHP1ThEnergyMWh,
	byHC1StateHC => byHC1StateHC,
	lrHC1OutTemp => lrHC1OutTemp,
	lrHC1OutTempAvg => lrHC1OutTempAvg,
	lrHC1RoomTemp => lrHC1RoomTemp,
	lrHC1SPRoomTemp => lrHC1SPRoomTemp,
	lrHC1PreFlowTemp => lrHC1PreFlowTemp,
	lrHC1SPFlowTemp => lrHC1SPFlowTemp);


fbHttpGet.bSend := FALSE;

FPDone(CLK:= bDone, Q=> );

fbClient.Execute();

//Error
IF fbHttpGet.bError OR fbClient.bError THEN bError := TRUE; ELSE bError := FALSE; END_IF	
	hrErrorCode := fbClient.hrErrorCode;

END_FUNCTION_BLOCK

// ---- FB/FB_OCHSNER_Web2Com2_Helper.TcPOU
FUNCTION_BLOCK FB_OCHSNER_Web2Com2_Helper
VAR_INPUT
	bSend				: BOOL;
END_VAR

VAR_IN_OUT
	fbClient			: FB_IotHttpClient;
END_VAR

VAR_OUTPUT
	bBusy				: BOOL;
	bError				: BOOL;
	byHP1StateHeatProd		: BYTE;
	lrHP1TWVtemp			: LREAL;
	lrHP1TWRtemp			: LREAL;
	lrHP1TQAtemp			: LREAL;
	lrHP1TQEtemp			: LREAL;
	lrHP1ThEnergykWh		: LREAL;
	lrHP1ThEnergyMWh		: LREAL;
	byHC1StateHC			: BYTE;
	lrHC1OutTemp			: LREAL;
	lrHC1OutTempAvg			: LREAL;
	lrHC1RoomTemp			: LREAL;
	lrHC1SPRoomTemp			: LREAL;
	lrHC1PreFlowTemp		: LREAL;
	lrHC1SPFlowTemp			: LREAL;
END_VAR

VAR
	fbRequest1			: FB_IotHttpRequest;
	fbRequest2			: FB_IotHttpRequest;

	fbJson				: FB_JsonDomParser;
	nState				: UDINT;
	RisingEdge			: R_TRIG;
	timTimeout			: TON;
	tTimeOut			: TIME := T#90S;
	bGetContentResult	: BOOL;
	sContent1			: STRING(511);
	sContent2			: STRING(511);
	
	bGetJsonResult		: BOOL;
	jsonDoc				: SJsonValue;
	jsonVal				: SJsonValue;
	
	nReqCount			: UDINT;	
	nResCount			: UDINT;
	nValidResCount		: UDINT;
	nErrCount			: UDINT;
END_VAR

//Timer for Timeout
timTimeout(IN:= nState = 1 AND bBusy, PT:= tTimeOut, Q=> , ET=> );
	IF timTimeout.Q THEN 
		nState := 0;
		bBusy := FALSE;
	END_IF

RisingEdge(CLK:= bSend );
CASE nState OF
0:	
	IF RisingEdge.Q THEN 
		IF 
			fbRequest1.SendRequest(sUri:='/web2com_2HP1.php', fbClient:=fbClient, eRequestType:=ETcIotHttpRequestType.HTTP_Get, 0, 0, 0) THEN				
			nState:= 1;
			nReqCount:= nReqCount+1;
			bBusy:= TRUE;
			bError:= FALSE;
		END_IF					
	END_IF
1:
	IF NOT fbRequest1.bBusy THEN
		bError:= TRUE;
		IF NOT fbRequest1.bError THEN				 
			bGetContentResult:= fbRequest1.GetContent(pContent:= ADR(sContent1), nContentSize:= SIZEOF(sContent1), bSetNullTermination:= TRUE);
			IF fbRequest1.nStatusCode >= 200 AND fbRequest1.nStatusCode < 300 THEN
				bGetJsonResult:= FALSE;
				jsonDoc:= fbRequest1.GetJsonDomContent(fbJson);
				IF jsonDoc <> 0 THEN
					bGetJsonResult:= TRUE;
					IF fbJson.HasMember(jsonDoc, '1211250')  THEN
						jsonVal:= fbJson.FindMember(jsonDoc, '1211250');
						nValidResCount:= nValidResCount+1;
						IF fbJson.IsNumber(jsonVal) THEN							
							byHP1StateHeatProd := DINT_TO_BYTE(fbJson.GetInt(jsonVal));									
						END_IF
						
						jsonVal:= fbJson.FindMember(jsonDoc, '1211251');
						nValidResCount:= nValidResCount+1;
						IF fbJson.IsDouble(jsonVal) THEN							
							lrHP1TWVtemp := fbJson.GetDouble(jsonVal);									
						END_IF
						
						jsonVal:= fbJson.FindMember(jsonDoc, '1211252');
						nValidResCount:= nValidResCount+1;
						IF fbJson.IsDouble(jsonVal) THEN							
							lrHP1TWRtemp := fbJson.GetDouble(jsonVal);									
						END_IF
						
						jsonVal:= fbJson.FindMember(jsonDoc, '1211253');
						nValidResCount:= nValidResCount+1;
						IF fbJson.IsDouble(jsonVal) THEN							
							lrHP1TQAtemp := fbJson.GetDouble(jsonVal);									
						END_IF
						
						jsonVal:= fbJson.FindMember(jsonDoc, '1211254');
						nValidResCount:= nValidResCount+1;
						IF fbJson.IsDouble(jsonVal) THEN							
							lrHP1TQEtemp := fbJson.GetDouble(jsonVal);									
						END_IF
						
						jsonVal:= fbJson.FindMember(jsonDoc, '1211258');
						nValidResCount:= nValidResCount+1;
						IF fbJson.IsNumber(jsonVal) THEN							
							lrHP1ThEnergykWh := fbJson.GetDouble(jsonVal);									
						END_IF
						
						jsonVal:= fbJson.FindMember(jsonDoc, '1211259');
						nValidResCount:= nValidResCount+1;
						IF fbJson.IsNumber(jsonVal) THEN							
							lrHP1ThEnergyMWh := fbJson.GetDouble(jsonVal);									
						END_IF
						
						bError:= FALSE;
						END_IF
					END_IF						
				nResCount:= nResCount+1;			
				END_IF
		END_IF
		(*
		IF NOT fbRequest2.bError THEN				 
			bGetContentResult:= fbRequest2.GetContent(pContent:= ADR(sContent2), nContentSize:= SIZEOF(sContent2), bSetNullTermination:= TRUE);
			IF fbRequest2.nStatusCode >= 200 AND fbRequest2.nStatusCode < 300 THEN
				bGetJsonResult:= FALSE;
				jsonDoc:= fbRequest2.GetJsonDomContent(fbJson);
				IF jsonDoc <> 0 THEN
					bGetJsonResult:= TRUE;
					IF fbJson.HasMember(jsonDoc, '1241190')  THEN
						jsonVal:= fbJson.FindMember(jsonDoc, '1241190');
						nValidResCount:= nValidResCount+1;
						IF fbJson.IsNumber(jsonVal) THEN							
							byHC1StateHC := DINT_TO_BYTE(fbJson.GetInt(jsonVal));									
						END_IF
						
						jsonVal:= fbJson.FindMember(jsonDoc, '1241191');
						nValidResCount:= nValidResCount+1;
						IF fbJson.IsDouble(jsonVal) THEN							
							lrHC1OutTemp := fbJson.GetDouble(jsonVal);									
						END_IF
						
						jsonVal:= fbJson.FindMember(jsonDoc, '1241192');
						nValidResCount:= nValidResCount+1;
						IF fbJson.IsDouble(jsonVal) THEN							
							lrHC1OutTempAvg := fbJson.GetDouble(jsonVal);									
						END_IF
						
						jsonVal:= fbJson.FindMember(jsonDoc, '1241193');
						nValidResCount:= nValidResCount+1;
						IF fbJson.IsDouble(jsonVal) THEN							
							lrHC1RoomTemp := fbJson.GetDouble(jsonVal);									
						END_IF
						
						jsonVal:= fbJson.FindMember(jsonDoc, '1241194');
						nValidResCount:= nValidResCount+1;
						IF fbJson.IsDouble(jsonVal) THEN							
							lrHC1SPRoomTemp := fbJson.GetDouble(jsonVal);									
						END_IF
						
						jsonVal:= fbJson.FindMember(jsonDoc, '1241195');
						nValidResCount:= nValidResCount+1;
						IF fbJson.IsDouble(jsonVal) THEN							
							lrHC1PreFlowTemp := fbJson.GetDouble(jsonVal);									
						END_IF
						
						jsonVal:= fbJson.FindMember(jsonDoc, '1241196');
						nValidResCount:= nValidResCount+1;
						IF fbJson.IsDouble(jsonVal) THEN							
							lrHC1SPFlowTemp := fbJson.GetDouble(jsonVal);									
						END_IF
						
						bError:= FALSE;
						END_IF
					END_IF						
				nResCount:= nResCount+1;			
				END_IF
		END_IF
		*)
		nState:= 0;
		bBusy:= FALSE;
		IF bError THEN
			nErrCount:= nErrCount+1;
		END_IF
	END_IF  	
END_CASE

END_FUNCTION_BLOCK

// ---- POUs/prgHP4.TcPOU
PROGRAM prgHP4
VAR
	fbWb2Com4						: FB_OCHSNER_Web2Com4;
	byHP1StateHeatProd		: BYTE;		//{#lynus.ag#()}
	lrHP1TWVtemp			: LREAL;	//{#lynus.ag#()}
	lrHP1TWRtemp			: LREAL;	//{#lynus.ag#()}
	lrHP1TQAtemp			: LREAL;	//{#lynus.ag#()}
	lrHP1TQEtemp			: LREAL;	//{#lynus.ag#()}
	lrHP1ThEnergykWh		: LREAL;	//{#lynus.ag#()}
	lrHP1ThEnergyMWh		: LREAL;	//{#lynus.ag#()}
	byHC1StateHC			: BYTE;		//{#lynus.ag#()}
	lrHC1OutTemp			: LREAL;	//{#lynus.ag#()}
	lrHC1OutTempAvg			: LREAL;	//{#lynus.ag#()}
	lrHC1SPRoomTemp			: LREAL;	//{#lynus.ag#()}
	lrHC1PreFlowTemp		: LREAL;	//{#lynus.ag#()}
	lrHC1SPFlowTemp			: LREAL;	//{#lynus.ag#()}
END_VAR

fbWb2Com4(
	bStart:= TRUE, 
	tDelayRequest:= T#60S, 
	sHostname:= 'localhost', 
	bValidResult=> , 
	bBusy=> , 
	bError=> , 
	bDone=> , 
	hrErrorCode=> ,
	byHP1StateHeatProd => byHP1StateHeatProd,
	lrHP1TWVtemp => lrHP1TWVtemp,
	lrHP1TWRtemp => lrHP1TWRtemp,
	lrHP1TQAtemp => lrHP1TQAtemp,
	lrHP1TQEtemp => lrHP1TQEtemp,
	lrHP1ThEnergykWh => lrHP1ThEnergykWh,
	lrHP1ThEnergyMWh => lrHP1ThEnergyMWh,
	byHC1StateHC => byHC1StateHC,
	lrHC1OutTemp => lrHC1OutTemp,
	lrHC1OutTempAvg => lrHC1OutTempAvg,
	lrHC1SPRoomTemp => lrHC1SPRoomTemp,
	lrHC1PreFlowTemp => lrHC1PreFlowTemp,
	lrHC1SPFlowTemp => lrHC1SPFlowTemp);

END_PROGRAM

// ---- FB/FB_OCHSNER_Web2Com4.TcPOU
FUNCTION_BLOCK FB_OCHSNER_Web2Com4
VAR_INPUT
	bStart				: BOOL;
	tDelayRequest		: TIME;		//Timer for delay before start with the next read or write Request
	sHostname			: STRING(255);		//Hostname or IP Adress from the Server
END_VAR

VAR_IN_OUT
END_VAR

VAR_OUTPUT
	bValidResult		: BOOL;							//Valid Result received from Server
    bBusy				: BOOL;							//Function is Busy
    bError				: BOOL;							//Error sucess
	bDone				: BOOL;							//True after the decoding from the received Json File
	bConnected			: BOOL;							//Connection to the Server
	hrErrorCode       	: HRESULT;						//Error Result from Http Client
	byHP1StateHeatProd		: BYTE;
	lrHP1TWVtemp			: LREAL;
	lrHP1TWRtemp			: LREAL;
	lrHP1TQAtemp			: LREAL;
	lrHP1TQEtemp			: LREAL;
	lrHP1ThEnergykWh		: LREAL;
	lrHP1ThEnergyMWh		: LREAL;
	byHC1StateHC			: BYTE;
	lrHC1OutTemp			: LREAL;
	lrHC1OutTempAvg			: LREAL;
	lrHC1RoomTemp			: LREAL;
	lrHC1SPRoomTemp			: LREAL;
	lrHC1PreFlowTemp		: LREAL;
	lrHC1SPFlowTemp			: LREAL;
END_VAR

VAR
	fbClient			: FB_IotHttpClient;
	fbHttpGet			: FB_OCHSNER_Web2Com4_Helper;
	timStartRequest		: TON;							//Timer to Start the Request
	FPStartRequest		: R_TRIG;						//Internal positive Edge
	FPDone				: R_TRIG;						//Internal positive Edge
	FNStart				: F_TRIG;						//Internal negative Edge
END_VAR

(*------------------------------------------------------------------------------------Configure HTTP Client------------------------------------------------------------------------------------------------------*)

fbClient.sHostName := sHostname;
fbClient.tConnectionTimeout := T#20S;
fbClient.bKeepAlive := FALSE;

IF NOT fbClient.bConfigured THEN 
	fbClient.nHostPort:= 80;
	fbClient.bKeepAlive := FALSE;
	fbClient.tConnectionTimeout := T#20S;
END_IF


//Timer to start the Request
FPStartRequest(CLK:= bStart, Q=> );
	timStartRequest(IN:= fbClient.bConfigured AND bStart AND NOT timStartRequest.Q, PT:= tDelayRequest, Q=> , ET=> );
		IF ((timStartRequest.Q AND NOT bBusy) OR (FPStartRequest.Q AND NOT bBusy AND fbClient.bConfigured)) THEN fbHttpGet.bSend := TRUE; END_IF

				
//Http Get Function
fbHttpGet(
	bSend:= , 
	fbClient:= fbClient, 
	bBusy=> bBusy, 
	bError=> ,
	byHP1StateHeatProd => byHP1StateHeatProd,
	lrHP1TWVtemp => lrHP1TWVtemp,
	lrHP1TWRtemp => lrHP1TWRtemp,
	lrHP1TQAtemp => lrHP1TQAtemp,
	lrHP1TQEtemp => lrHP1TQEtemp,
	lrHP1ThEnergykWh => lrHP1ThEnergykWh,
	lrHP1ThEnergyMWh => lrHP1ThEnergyMWh,
	byHC1StateHC => byHC1StateHC,
	lrHC1OutTemp => lrHC1OutTemp,
	lrHC1OutTempAvg => lrHC1OutTempAvg,
	lrHC1SPRoomTemp => lrHC1SPRoomTemp,
	lrHC1PreFlowTemp => lrHC1PreFlowTemp,
	lrHC1SPFlowTemp => lrHC1SPFlowTemp);


fbHttpGet.bSend := FALSE;

FPDone(CLK:= bDone, Q=> );

fbClient.Execute();

//Error
IF fbHttpGet.bError OR fbClient.bError THEN bError := TRUE; ELSE bError := FALSE; END_IF	
	hrErrorCode := fbClient.hrErrorCode;

END_FUNCTION_BLOCK

// ---- FB/FB_OCHSNER_Web2Com4_Helper.TcPOU
FUNCTION_BLOCK FB_OCHSNER_Web2Com4_Helper
VAR_INPUT
	bSend				: BOOL;
END_VAR

VAR_IN_OUT
	fbClient			: FB_IotHttpClient;
END_VAR

VAR_OUTPUT
	bBusy				: BOOL;
	bError				: BOOL;
	byHP1StateHeatProd		: BYTE;
	lrHP1TWVtemp			: LREAL;
	lrHP1TWRtemp			: LREAL;
	lrHP1TQAtemp			: LREAL;
	lrHP1TQEtemp			: LREAL;
	lrHP1ThEnergykWh		: LREAL;
	lrHP1ThEnergyMWh		: LREAL;
	byHC1StateHC			: BYTE;
	lrHC1OutTemp			: LREAL;
	lrHC1OutTempAvg			: LREAL;
	lrHC1SPRoomTemp			: LREAL;
	lrHC1PreFlowTemp		: LREAL;
	lrHC1SPFlowTemp			: LREAL;
END_VAR

VAR
	fbRequest1			: FB_IotHttpRequest;
	fbRequest2			: FB_IotHttpRequest;

	fbJson				: FB_JsonDomParser;
	nState				: UDINT;
	RisingEdge			: R_TRIG;
	timTimeout			: TON;
	tTimeOut			: TIME := T#90S;
	bGetContentResult	: BOOL;
	sContent1			: STRING(511);
	sContent2			: STRING(511);
	
	bGetJsonResult		: BOOL;
	jsonDoc				: SJsonValue;
	jsonVal				: SJsonValue;
	
	nReqCount			: UDINT;	
	nResCount			: UDINT;
	nValidResCount		: UDINT;
	nErrCount			: UDINT;
END_VAR

//Timer for Timeout
timTimeout(IN:= nState = 1 AND bBusy, PT:= tTimeOut, Q=> , ET=> );
	IF timTimeout.Q THEN 
		nState := 0;
		bBusy := FALSE;
	END_IF

RisingEdge(CLK:= bSend );
CASE nState OF
0:	
	IF RisingEdge.Q THEN 
		IF 
			fbRequest1.SendRequest(sUri:='/web2com_4HP1.php', fbClient:=fbClient, eRequestType:=ETcIotHttpRequestType.HTTP_Get, 0, 0, 0) AND
			fbRequest2.SendRequest(sUri:='/web2com_4HC1.php', fbClient:=fbClient, eRequestType:=ETcIotHttpRequestType.HTTP_Get, 0, 0, 0) THEN				
			nState:= 1;
			nReqCount:= nReqCount+1;
			bBusy:= TRUE;
			bError:= FALSE;
		END_IF					
	END_IF
1:
	IF NOT fbRequest1.bBusy AND NOT fbRequest2.bBusy THEN
		bError:= TRUE;
		IF NOT fbRequest1.bError THEN				 
			bGetContentResult:= fbRequest1.GetContent(pContent:= ADR(sContent1), nContentSize:= SIZEOF(sContent1), bSetNullTermination:= TRUE);
			IF fbRequest1.nStatusCode >= 200 AND fbRequest1.nStatusCode < 300 THEN
				bGetJsonResult:= FALSE;
				jsonDoc:= fbRequest1.GetJsonDomContent(fbJson);
				IF jsonDoc <> 0 THEN
					bGetJsonResult:= TRUE;
					IF fbJson.HasMember(jsonDoc, '1211250')  THEN
						jsonVal:= fbJson.FindMember(jsonDoc, '1211250');
						nValidResCount:= nValidResCount+1;
						IF fbJson.IsNumber(jsonVal) THEN							
							byHP1StateHeatProd := DINT_TO_BYTE(fbJson.GetInt(jsonVal));									
						END_IF
						
						jsonVal:= fbJson.FindMember(jsonDoc, '1211251');
						nValidResCount:= nValidResCount+1;
						IF fbJson.IsDouble(jsonVal) THEN							
							lrHP1TWVtemp := fbJson.GetDouble(jsonVal);									
						END_IF
						
						jsonVal:= fbJson.FindMember(jsonDoc, '1211253');
						nValidResCount:= nValidResCount+1;
						IF fbJson.IsDouble(jsonVal) THEN							
							lrHP1TWRtemp := fbJson.GetDouble(jsonVal);									
						END_IF
						
						jsonVal:= fbJson.FindMember(jsonDoc, '1211254');
						nValidResCount:= nValidResCount+1;
						IF fbJson.IsDouble(jsonVal) THEN							
							lrHP1TQAtemp := fbJson.GetDouble(jsonVal);									
						END_IF
						
						jsonVal:= fbJson.FindMember(jsonDoc, '1211255');
						nValidResCount:= nValidResCount+1;
						IF fbJson.IsDouble(jsonVal) THEN							
							lrHP1TQEtemp := fbJson.GetDouble(jsonVal);									
						END_IF
						
						jsonVal:= fbJson.FindMember(jsonDoc, '1211258');
						nValidResCount:= nValidResCount+1;
						IF fbJson.IsNumber(jsonVal) THEN							
							lrHP1ThEnergykWh := fbJson.GetDouble(jsonVal);									
						END_IF
						
						jsonVal:= fbJson.FindMember(jsonDoc, '1211259');
						nValidResCount:= nValidResCount+1;
						IF fbJson.IsNumber(jsonVal) THEN							
							lrHP1ThEnergyMWh := fbJson.GetDouble(jsonVal);									
						END_IF
						
						bError:= FALSE;
						END_IF
					END_IF						
				nResCount:= nResCount+1;			
				END_IF
		END_IF
		
		IF NOT fbRequest2.bError THEN				 
			bGetContentResult:= fbRequest2.GetContent(pContent:= ADR(sContent2), nContentSize:= SIZEOF(sContent2), bSetNullTermination:= TRUE);
			IF fbRequest2.nStatusCode >= 200 AND fbRequest2.nStatusCode < 300 THEN
				bGetJsonResult:= FALSE;
				jsonDoc:= fbRequest2.GetJsonDomContent(fbJson);
				IF jsonDoc <> 0 THEN
					bGetJsonResult:= TRUE;
					IF fbJson.HasMember(jsonDoc, '1241190')  THEN
						jsonVal:= fbJson.FindMember(jsonDoc, '1241190');
						nValidResCount:= nValidResCount+1;
						IF fbJson.IsNumber(jsonVal) THEN							
							byHC1StateHC := DINT_TO_BYTE(fbJson.GetInt(jsonVal));									
						END_IF
						
						jsonVal:= fbJson.FindMember(jsonDoc, '1241191');
						nValidResCount:= nValidResCount+1;
						IF fbJson.IsDouble(jsonVal) THEN							
							lrHC1OutTemp := fbJson.GetDouble(jsonVal);									
						END_IF
						
						jsonVal:= fbJson.FindMember(jsonDoc, '1241192');
						nValidResCount:= nValidResCount+1;
						IF fbJson.IsDouble(jsonVal) THEN							
							lrHC1OutTempAvg := fbJson.GetDouble(jsonVal);									
						END_IF
			
						jsonVal:= fbJson.FindMember(jsonDoc, '1241193');
						nValidResCount:= nValidResCount+1;
						IF fbJson.IsDouble(jsonVal) THEN							
							lrHC1SPRoomTemp := fbJson.GetDouble(jsonVal);									
						END_IF
						
						jsonVal:= fbJson.FindMember(jsonDoc, '1241194');
						nValidResCount:= nValidResCount+1;
						IF fbJson.IsDouble(jsonVal) THEN							
							lrHC1PreFlowTemp := fbJson.GetDouble(jsonVal);									
						END_IF
						
						jsonVal:= fbJson.FindMember(jsonDoc, '1241195');
						nValidResCount:= nValidResCount+1;
						IF fbJson.IsDouble(jsonVal) THEN							
							lrHC1SPFlowTemp := fbJson.GetDouble(jsonVal);									
						END_IF
						
						bError:= FALSE;
						END_IF
					END_IF						
				nResCount:= nResCount+1;			
				END_IF
		END_IF
		
		nState:= 0;
		bBusy:= FALSE;
		IF bError THEN
			nErrCount:= nErrCount+1;
		END_IF
	END_IF  	
END_CASE

END_FUNCTION_BLOCK

// ---- POUs/prgPV.TcPOU
PROGRAM prgPV
VAR
	fbPVCounter1		: FB_EnergyCounter;
	fbPVCounter2		: FB_EnergyCounter;
	lrPowerPV1			: LREAL;				//{#lynus.ag#()}
	lrPowerPV2			: LREAL;				//{#lynus.ag#()}
	lrPowerPVTotal		: LREAL;				//{#lynus.ag#()}
	byErrorWarningPV	: BYTE;					//{#lynus.ag#()}
	FB_PV1:FB_TCPModbusRequest_PV;
	FB_PV2:FB_TCPModbusRequest_PV;
	lrVoltagePV1_L1L2_V		: LREAL;				//{#lynus.ag#()}
	lrVoltagePV1_L2L3_V		: LREAL;				//{#lynus.ag#()}
	lrVoltagePV1_L3L1_V		: LREAL;				//{#lynus.ag#()}
	lrVoltagePV2_L1L2_V		: LREAL;				//{#lynus.ag#()}
	lrVoltagePV2_L2L3_V		: LREAL;				//{#lynus.ag#()}
	lrVoltagePV2_L3L1_V		: LREAL;				//{#lynus.ag#()}
END_VAR
VAR PERSISTENT
	lrCounterPV1		: LREAL;					//{#lynus.ag#()}
	lrCounterPV2		: LREAL;					//{#lynus.ag#()}
	lrCounterPVTotal	: LREAL;					//{#lynus.ag#()}
END_VAR


FB_PV1	(	b_Enable:= TRUE, 
			str_IPAdress:= '192.168.11.171', 
			lreal_RealPower_kW=> lrPowerPV1,
			lreal_Voltage_L1L2_V=> lrVoltagePV1_L1L2_V , 
			lreal_Voltage_L2L3_V=> lrVoltagePV1_L2L3_V , 
			lreal_Voltage_L3L1_V=> lrVoltagePV1_L3L1_V);


fbPVCounter1(	byActiveTariff := 1,	
				lrPowerInput := 0-lrPowerPV1,
				lrTotalCounterEnergy_Production => lrCounterPV1);
	

FB_PV2	(	b_Enable:= TRUE, 
			str_IPAdress:= '192.168.11.172', 
			lreal_RealPower_kW=> lrPowerPV2,
			lreal_Voltage_L1L2_V=> lrVoltagePV2_L1L2_V , 
			lreal_Voltage_L2L3_V=> lrVoltagePV2_L2L3_V , 
			lreal_Voltage_L3L1_V=> lrVoltagePV2_L3L1_V);

fbPVCounter2(	byActiveTariff := 1,	
				lrPowerInput := 0-lrPowerPV2,
				lrTotalCounterEnergy_Production => lrCounterPV2);
	
lrPowerPVTotal := lrPowerPV1 + lrPowerPV2;
lrCounterPVTotal := lrCounterPV1 + lrCounterPV2;

END_PROGRAM

// ---- FB/FB_TCPModbusRequest_PV.TcPOU
FUNCTION_BLOCK FB_TCPModbusRequest_PV
VAR_INPUT
	b_Enable: BOOL;
	str_IPAdress: STRING(15);
	
		
END_VAR
VAR_OUTPUT

	lreal_RealPower_kW:LREAL;
	lreal_Voltage_L1L2_V: LREAL;
	lreal_Voltage_L2L3_V: LREAL;
	lreal_Voltage_L3L1_V: LREAL;
	lreal_Voltage_L1_V: LREAL;
	lreal_Voltage_L2_V: LREAL;
	lreal_Voltage_L3_V: LREAL;
	lreal_Current_L1_A: LREAL;
	lreal_Current_L2_A: LREAL;
	lreal_Current_L3_A: LREAL;
	lreal_PeakPowerDay_kW: LREAL;
	lreal_Power2_kW: LREAL;
	lreal_ReactivePower_kVAr: LREAL;
	lreal_PowerFactor: LREAL;
	lreal_Frequency_Hz: LREAL;
	lreal_Efficiency: LREAL;
	lreal_InternalTemperature_C: LREAL;
	lreal_IsolationResistance_MOhm: LREAL;
END_VAR
VAR
	i_State:INT;
	FB_SocketConnect : FB_SocketConnect;
	hSocket : T_HSOCKET;
	FB_SocketSend : FB_SocketSend;
	FB_SocketReceive : FB_SocketReceive;
	byteSendString : ARRAY[1..12] OF BYTE;
	FB_CloseSockets: FB_SocketCloseAll;
	
	ton_TimeOut: Ton;
	ton_WaitforReconnect: Ton;
	ton_ConnectionEstablised: Ton;
	time_ReconnectTime:TIME:=T#30M;
	b_configured: BOOL;
	byteReceiveString : ARRAY[1..200] OF BYTE;
	FB_BYTE_TO_WORD_1 : FB_CV_BYTE_TO_WORD;
	FB_BYTE_TO_WORD_2 : FB_CV_BYTE_TO_WORD;
	FB_WORD_TO_INT : FB_CV_WORD_TO_INT;
	ton_WaitforNetxtRequest: Ton;
	ton_Wait: Ton;
	int_SuccessCounter: INT;
	int_ReconnectCounter: INT;
	int_ErrorCount: INT;
	fbConvertWordToDword		: FB_CV_WORD_TO_DWORD;			//Convert Word to Dword
	fb_ConvertBytesToLreal		:fb_Convert4BytesToLreal;

END_VAR





IF NOT b_Enable THEN			// go to state 0 if not enabled
	i_State := 0;
END_IF


CASE i_State OF
	0:	// wait for enable state
		IF b_Enable THEN
			i_State := 1;
		END_IF
		FB_SocketConnect.bExecute := FALSE;
		FB_SocketSend.bExecute := FALSE;
		FB_SocketSend.bExecute := FALSE;
		ton_TimeOut.IN :=FALSE;	
		ton_ConnectionEstablised.IN := FALSE;
	

	1: // check if configured
		IF b_configured = FALSE THEN
			// request FC3, Register 32064, 25 Words --> Real PV Power ff
			byteSendString[1] := 0;
			byteSendString[2] := 1;
			byteSendString[3] := 0;
			byteSendString[4] := 0;
			byteSendString[5] := 0;
			byteSendString[6] := 6;
			byteSendString[7] := 1;
			byteSendString[8] := 3;
			byteSendString[9] := 125;
			byteSendString[10] := 64;
			byteSendString[11] := 0;
			byteSendString[12] := 25;
		
			b_configured := TRUE;
		END_IF
		i_State := i_State+1;
		
	2: // open socket
		FB_SocketConnect.bExecute := TRUE;
		ton_TimeOut.IN :=TRUE;
		i_State := i_State+1;
		
	3: // wait for connection established	
		IF NOT FB_SocketConnect.bBusy AND NOT FB_SocketConnect.bError THEN
			ton_TimeOut.IN :=FALSE;
			ton_ConnectionEstablised.IN := TRUE;
			i_State := i_State+1;
		ELSIF FB_SocketConnect.bError OR ton_TimeOut.Q THEN
			ton_TimeOut.IN :=FALSE;
			i_State := 100;
		END_IF
	
	4: //connection established, request data
		ton_Wait.IN := TRUE;
		IF ton_Wait.Q THEN
			FB_SocketSend.bExecute := TRUE;
			ton_TimeOut.IN :=TRUE;
			ton_Wait.IN := FALSE;
			i_State := i_State+1;
		END_IF
	
	5: // wait for request sent
		IF NOT FB_SocketSend.bBusy AND NOT FB_SocketSend.bError THEN
			ton_TimeOut.IN :=FALSE;
			FB_SocketSend.bExecute := FALSE;
			i_State := i_State+1;  
		ELSIF FB_SocketSend.bError OR ton_TimeOut.Q THEN
			FB_SocketSend.bExecute := FALSE;
			ton_TimeOut.IN :=FALSE;
			i_State := 100;
		END_IF
		
	6: // wait for data
		ton_Wait.IN := TRUE;
		IF ton_Wait.Q THEN
			FB_SocketReceive.bExecute := TRUE;
			ton_Wait.IN := FALSE;
			i_State := i_State+1; 
		END_IF		 
	
	7:	
		ton_Wait.IN := TRUE;
		IF ton_Wait.Q THEN
			ton_TimeOut.IN :=TRUE;
			i_State := i_State+1; 
		END_IF	
	
	8: // convert received data
		IF NOT FB_SocketReceive.bBusy AND NOT FB_SocketReceive.bError THEN
			int_SuccessCounter := int_SuccessCounter+1;
			ton_TimeOut.IN :=FALSE;
			FB_SocketReceive.bExecute := FALSE;
	
			FB_BYTE_TO_WORD_1(byInputValue_1 := byteReceiveString[14],byInputValue_2 := byteReceiveString[15], Ebyteorderforconvert := Ebyteorder.EBIGENDIAN, woutputvalue => );
			lreal_Voltage_L1L2_V := WORD_TO_LREAL(FB_BYTE_TO_WORD_1.woutputvalue)/10;
			FB_BYTE_TO_WORD_1(byInputValue_1 := byteReceiveString[16],byInputValue_2 := byteReceiveString[17], Ebyteorderforconvert := Ebyteorder.EBIGENDIAN, woutputvalue => );
			lreal_Voltage_L2L3_V := WORD_TO_LREAL(FB_BYTE_TO_WORD_1.woutputvalue)/10;
			FB_BYTE_TO_WORD_1(byInputValue_1 := byteReceiveString[18],byInputValue_2 := byteReceiveString[19], Ebyteorderforconvert := Ebyteorder.EBIGENDIAN, woutputvalue => );
			lreal_Voltage_L3L1_V := WORD_TO_LREAL(FB_BYTE_TO_WORD_1.woutputvalue)/10;
			FB_BYTE_TO_WORD_1(byInputValue_1 := byteReceiveString[20],byInputValue_2 := byteReceiveString[21], Ebyteorderforconvert := Ebyteorder.EBIGENDIAN, woutputvalue => );
			lreal_Voltage_L1_V := WORD_TO_LREAL(FB_BYTE_TO_WORD_1.woutputvalue)/10;
			FB_BYTE_TO_WORD_1(byInputValue_1 := byteReceiveString[22],byInputValue_2 := byteReceiveString[23], Ebyteorderforconvert := Ebyteorder.EBIGENDIAN, woutputvalue => );
			lreal_Voltage_L2_V := WORD_TO_LREAL(FB_BYTE_TO_WORD_1.woutputvalue)/10;
			FB_BYTE_TO_WORD_1(byInputValue_1 := byteReceiveString[24],byInputValue_2 := byteReceiveString[25], Ebyteorderforconvert := Ebyteorder.EBIGENDIAN, woutputvalue => );
			lreal_Voltage_L3_V := WORD_TO_LREAL(FB_BYTE_TO_WORD_1.woutputvalue)/10;


			fb_ConvertBytesToLreal(	by_InputValue_1:= byteReceiveString[10], 
									by_InputValue_2:= byteReceiveString[11], 
									by_InputValue_3:= byteReceiveString[12], 
									by_InputValue_4:= byteReceiveString[13], 
									int_Divider:= 1000, 
									lreal_Output=> lreal_RealPower_kW);

			fb_ConvertBytesToLreal(	by_InputValue_1:= byteReceiveString[26], 
									by_InputValue_2:= byteReceiveString[27], 
									by_InputValue_3:= byteReceiveString[28], 
									by_InputValue_4:= byteReceiveString[29], 
									int_Divider:= 1000, 
									lreal_Output=> lreal_Current_L1_A);
									
			fb_ConvertBytesToLreal(	by_InputValue_1:= byteReceiveString[30], 
									by_InputValue_2:= byteReceiveString[31], 
									by_InputValue_3:= byteReceiveString[32], 
									by_InputValue_4:= byteReceiveString[33], 
									int_Divider:= 1000, 
									lreal_Output=> lreal_Current_L2_A);

			fb_ConvertBytesToLreal(	by_InputValue_1:= byteReceiveString[34], 
									by_InputValue_2:= byteReceiveString[35], 
									by_InputValue_3:= byteReceiveString[36], 
									by_InputValue_4:= byteReceiveString[37], 
									int_Divider:= 1000, 
									lreal_Output=> lreal_Current_L3_A);
									
			fb_ConvertBytesToLreal(	by_InputValue_1:= byteReceiveString[38], 
									by_InputValue_2:= byteReceiveString[39], 
									by_InputValue_3:= byteReceiveString[40], 
									by_InputValue_4:= byteReceiveString[41], 
									int_Divider:= 1000, 
									lreal_Output=> lreal_PeakPowerDay_kW );

			fb_ConvertBytesToLreal(	by_InputValue_1:= byteReceiveString[42], 
									by_InputValue_2:= byteReceiveString[43], 
									by_InputValue_3:= byteReceiveString[44], 
									by_InputValue_4:= byteReceiveString[45], 
									int_Divider:= 1000, 
									lreal_Output=> lreal_Power2_kW);
			
			fb_ConvertBytesToLreal(	by_InputValue_1:= byteReceiveString[46], 
									by_InputValue_2:= byteReceiveString[47], 
									by_InputValue_3:= byteReceiveString[48], 
									by_InputValue_4:= byteReceiveString[49], 
									int_Divider:= 1000, 
									lreal_Output=>lreal_ReactivePower_kVAr );

			FB_BYTE_TO_WORD_1(byInputValue_1 := byteReceiveString[50],byInputValue_2 := byteReceiveString[51], Ebyteorderforconvert := Ebyteorder.EBIGENDIAN, woutputvalue => );
			lreal_PowerFactor := WORD_TO_LREAL(FB_BYTE_TO_WORD_1.woutputvalue)/1000;
			FB_BYTE_TO_WORD_1(byInputValue_1 := byteReceiveString[52],byInputValue_2 := byteReceiveString[53], Ebyteorderforconvert := Ebyteorder.EBIGENDIAN, woutputvalue => );
			lreal_Frequency_Hz := WORD_TO_LREAL(FB_BYTE_TO_WORD_1.woutputvalue)/100;
			FB_BYTE_TO_WORD_1(byInputValue_1 := byteReceiveString[54],byInputValue_2 := byteReceiveString[55], Ebyteorderforconvert := Ebyteorder.EBIGENDIAN, woutputvalue => );
			lreal_Efficiency := WORD_TO_LREAL(FB_BYTE_TO_WORD_1.woutputvalue)/100;
			FB_BYTE_TO_WORD_1(byInputValue_1 := byteReceiveString[56],byInputValue_2 := byteReceiveString[57], Ebyteorderforconvert := Ebyteorder.EBIGENDIAN, woutputvalue => );
			lreal_InternalTemperature_C := WORD_TO_LREAL(FB_BYTE_TO_WORD_1.woutputvalue)/10;
			FB_BYTE_TO_WORD_1(byInputValue_1 := byteReceiveString[58],byInputValue_2 := byteReceiveString[59], Ebyteorderforconvert := Ebyteorder.EBIGENDIAN, woutputvalue => );
			lreal_IsolationResistance_MOhm := WORD_TO_LREAL(FB_BYTE_TO_WORD_1.woutputvalue)/1000;

		
			//FB_WORD_TO_INT(wInputValue := FB_BYTE_TO_WORD.woutputvalue, iOutputValue => );
			//lreal_RealPower_kW := (INT_TO_LREAL(FB_WORD_TO_INT.iOutputValue))/1000;

			i_State := i_State+1;
		ELSIF FB_SocketSend.bError OR ton_TimeOut.Q THEN
 			FB_SocketReceive.bExecute := FALSE;
			ton_TimeOut.IN :=FALSE;
			i_State := 100;
		END_IF
	
	9: // for for next request
		ton_WaitforNetxtRequest.IN := TRUE;
		IF NOT b_Enable THEN
			ton_WaitforNetxtRequest.IN := FALSE;
			i_State := 10;
		END_IF
		IF ton_WaitforNetxtRequest.Q THEN
			ton_WaitforNetxtRequest.IN := FALSE;
			i_State := 4;
		END_IF
		IF 	ton_ConnectionEstablised.Q THEN 
			ton_WaitforNetxtRequest.IN := FALSE;
			i_State := 10;
		END_IF

	10: // close sockets
		FB_CloseSockets.bExecute := TRUE;
		ton_TimeOut.IN :=TRUE;
		i_State := i_State+1;
		
	11: // wait for sockets closed
		
		IF NOT FB_CloseSockets.bBusy THEN
			int_ReconnectCounter := int_ReconnectCounter+1;
			FB_CloseSockets.bExecute := FALSE;
			i_State := 0;
		ELSIF FB_CloseSockets.bError THEN
			int_ReconnectCounter := int_ReconnectCounter+1;
			FB_CloseSockets.bExecute := FALSE;
			i_State := 0;
		END_IF

	100: // wait state for reconect
		
		FB_SocketConnect.bExecute := FALSE;
		FB_SocketSend.bExecute := FALSE;
		FB_SocketReceive.bExecute := FALSE;
		ton_ConnectionEstablised.IN := FALSE;
		ton_TimeOut.IN :=FALSE;
		ton_WaitforReconnect.IN := TRUE;
		IF ton_WaitforReconnect.Q THEN
			int_ErrorCount := int_ErrorCount+1;
			ton_WaitforReconnect.IN := FALSE;
			i_State := 10;
		END_IF
	
END_CASE



FB_SocketConnect(
	sSrvNetId := '',
	sRemoteHost := str_IPAdress,
	nRemotePort := 502,
	bExecute := ,
	tTimeout := T#1S,
	bBusy =>,
	bError =>,
	nErrId =>,
	hSocket => hSocket);
	
FB_SocketSend(
	sSrvNetId:= '', 
	hSocket:= hSocket, 
	cbLen:= 12,
	pSrc:= ADR( byteSendString ), 
	bExecute:= , 
	tTimeout:= T#3S, 
	bBusy=> , 
	bError=> , 
	nErrId=> );
	
FB_SocketReceive(
	sSrvNetId:= '', 
	hSocket:= hSocket, 
	cbLen:= 200, 
	pDest:= ADR( byteReceiveString ), 
	bExecute:= , 
	tTimeout:= T#3S, 
	bBusy=> , 
	bError=> , 
	nErrId=> , 
	nRecBytes=> );

FB_CloseSockets(
	sSrvNetId:= '', 
	bExecute:= , 
	tTimeout:= T#2S, 
	bBusy=> , 
	bError=> , 
	nErrId=> );
	
ton_TimeOut(PT := T#5S);
ton_WaitforReconnect(PT := T#10S);
ton_ConnectionEstablised(pt := time_ReconnectTime);
ton_WaitforNetxtRequest(PT:= T#10S);
ton_Wait(PT:=T#2S);

END_FUNCTION_BLOCK

// ---- FB/fb_Convert4BytesToLreal.TcPOU
FUNCTION_BLOCK fb_Convert4BytesToLreal
VAR_INPUT
	by_InputValue_1:BYTE;
	by_InputValue_2:BYTE;
	by_InputValue_3:BYTE;
	by_InputValue_4:BYTE;
	int_Divider: INT;
END_VAR
VAR_OUTPUT
	lreal_Output:LREAL;
END_VAR
VAR
	FB_BYTE_TO_WORD_1 : FB_CV_BYTE_TO_WORD;
	FB_BYTE_TO_WORD_2 : FB_CV_BYTE_TO_WORD;
	fbConvertWordToDword		: FB_CV_WORD_TO_DWORD;			//Convert Word to Dword

END_VAR

IF int_Divider =0 THEN
	int_Divider :=1;
END_IF
FB_BYTE_TO_WORD_1(byInputValue_1 := by_InputValue_1,byInputValue_2 := by_InputValue_2, Ebyteorderforconvert := Ebyteorder.ebigENDIAN, woutputvalue => );
FB_BYTE_TO_WORD_2(byInputValue_1 := by_InputValue_3,byInputValue_2 := by_InputValue_4, Ebyteorderforconvert := Ebyteorder.ebigENDIAN, woutputvalue => );

fbConvertWordToDword(wInputValue_1:= FB_BYTE_TO_WORD_1.woutputvalue, wInputValue_2:= FB_BYTE_TO_WORD_2.woutputvalue, eByteOrderForConvert:= eByteOrder.eBigEndian , dwOutputValue=> );
lreal_Output :=DINT_TO_LREAL( DWORD_TO_DINT(fbConvertWordToDword.dwOutputValue))/int_Divider;

END_FUNCTION_BLOCK

// ---- POUs/prgPersistent.TcPOU
PROGRAM prgPersistent
VAR
	fbUSV		: FB_WritePersistentData_General;
	fb_Reboot: NT_Reboot;
	mReboot: BOOL:=FALSE;
	ton_liveCount: Ton;
	int_LiveCount: INT;										//{#lynus.ag#()}
END_VAR

fbUSV(
	eSaveModeData:= eUSVSaveMode.eSaveWhenPowerfail, 
	bLoadPersistentDataOk=> , 
	bError=> , 
	bySaveProcess=> , 
	dwStorageLast24h=> , 
	udiErrorCode=> );


fb_Reboot (
	netid := '',
	delay := 5,
	start := mReboot);
	

ton_liveCount( 	IN := NOT ton_liveCount.Q,
				PT := T#1M);
				
IF ton_liveCount.Q THEN
	int_LiveCount := int_LiveCount+1;	
END_IF

END_PROGRAM

// ---- POUs/prgComEffIO.TcPOU
PROGRAM prgComEffIO
VAR
	fbCom			: FB_MqttCommunicator_V2;
END_VAR


fbCom(
	bConnect:= TRUE, 
	strAuthKey:= 'BE736352867778' , 
	sUserName:= 'ee550063-1f43-4a46-bb0f-f5150fb59b57', 
	sUserPassword:= 'f17bd22e-1272-413e-8784-0472919c203c' , 
	eSavePositionCertificate:= eSavePositionOnPLC.ePostionC , 
	time_HeartBeat_sec:= , 
	bConnected=> , 
	bError=> , 
	hrErrorCode=> , 
	eConnectionState=> , 
	eErrorMessage_Out=> );
	
(*
fbCom(
	bConnect:= TRUE, 
	strAuthKey:= 'EIO08031879806' , 
	sUserName:= '02a135c3-ecb9-49f0-8ebf-5a80a42f4424', 
	sUserPassword:= 'ff07c9b9-2bd2-49ce-ac0e-e8974bf50ecc' , 
	eSavePositionCertificate:= eSavePositionOnPLC.ePostionC , 
	time_HeartBeat_sec:= , 
	bConnected=> , 
	bError=> , 
	hrErrorCode=> , 
	eConnectionState=> , 
	eErrorMessage_Out=> );
*)

END_PROGRAM

// ---- FB/FB_TCPModbusRequest_Grid.TcPOU
FUNCTION_BLOCK FB_TCPModbusRequest_Grid
VAR_INPUT
	b_Enable: BOOL;
	str_IPAdress: STRING(15);
	
		
END_VAR
VAR_OUTPUT
	b_MeterOnline: BOOL;
	lreal_GridVoltage_L1L2_V: LREAL;
	lreal_GridVoltage_L2L3_V: LREAL;
	lreal_GridVoltage_L3L1_V: LREAL;
	lreal_GridVoltage_L1_V: LREAL;
	lreal_GridVoltage_L2_V: LREAL;
	lreal_GridVoltage_L3_V: LREAL;
	lreal_GridCurrent_L1_A: LREAL;
	lreal_GridCurrent_L2_A: LREAL;
	lreal_GridCurrent_L3_A: LREAL;
	lreal_GridPower_kW: LREAL;
	lreal_GridReactivePower_kVAr: LREAL;
	lreal_GridPowerFactor: LREAL;
	lreal_GridFrequency_Hz: LREAL;
	lreal_GridEnergyDelivered_kWh: LREAL;
	lreal_GridEnergySupllied_kWh: LREAL;
END_VAR
VAR
	i_State:INT;
	FB_SocketConnect : FB_SocketConnect;
	hSocket : T_HSOCKET;
	FB_SocketSend : FB_SocketSend;
	FB_SocketReceive : FB_SocketReceive;
	byteSendString : ARRAY[1..12] OF BYTE;
	FB_CloseSockets: FB_SocketCloseAll;
	
	ton_TimeOut: Ton;
	ton_WaitforReconnect: Ton;
	ton_ConnectionEstablised: Ton;
	time_ReconnectTime:TIME:=T#30M;
	b_configured: BOOL;
	byteReceiveString : ARRAY[1..200] OF BYTE;
	FB_BYTE_TO_WORD_1 : FB_CV_BYTE_TO_WORD;
	FB_BYTE_TO_WORD_2 : FB_CV_BYTE_TO_WORD;
	FB_WORD_TO_INT : FB_CV_WORD_TO_INT;
	ton_WaitforNetxtRequest: Ton;
	ton_Wait: Ton;
	int_SuccessCounter: INT;
	int_ReconnectCounter: INT;
	int_ErrorCount: INT;
	fbConvertWordToDword		: FB_CV_WORD_TO_DWORD;			//Convert Word to Dword
	fb_ConvertBytesToLreal		:fb_Convert4BytesToLreal;

END_VAR





IF NOT b_Enable THEN			// go to state 0 if not enabled
	i_State := 0;
END_IF


CASE i_State OF
	0:	// wait for enable state
		IF b_Enable THEN
			i_State := 1;
		END_IF
		FB_SocketConnect.bExecute := FALSE;
		FB_SocketSend.bExecute := FALSE;
		FB_SocketSend.bExecute := FALSE;
		ton_TimeOut.IN :=FALSE;	
		ton_ConnectionEstablised.IN := FALSE;
	

	1: // check if configured
		IF b_configured = FALSE THEN
			// request FC3, Register 37100 16#90EC, 38 Words 
			byteSendString[1] := 0;
			byteSendString[2] := 1;
			byteSendString[3] := 0;
			byteSendString[4] := 0;
			byteSendString[5] := 0;
			byteSendString[6] := 6;
			byteSendString[7] := 1;
			byteSendString[8] := 3;
			byteSendString[9] := 16#90;
			byteSendString[10] := 16#EC;
			byteSendString[11] := 0;
			byteSendString[12] := 38;
			b_configured := TRUE;
		END_IF
		i_State := i_State+1;
		
	2: // open socket
		FB_SocketConnect.bExecute := TRUE;
		ton_TimeOut.IN :=TRUE;
		i_State := i_State+1;
		
	3: // wait for connection established	
		IF NOT FB_SocketConnect.bBusy AND NOT FB_SocketConnect.bError THEN
			ton_TimeOut.IN :=FALSE;
			ton_ConnectionEstablised.IN := TRUE;
			i_State := i_State+1;
		ELSIF FB_SocketConnect.bError OR ton_TimeOut.Q THEN
			ton_TimeOut.IN :=FALSE;
			i_State := 100;
		END_IF
	
	4: //connection established, request data
		ton_Wait.IN := TRUE;
		IF ton_Wait.Q THEN
			FB_SocketSend.bExecute := TRUE;
			ton_TimeOut.IN :=TRUE;
			ton_Wait.IN := FALSE;
			i_State := i_State+1;
		END_IF
	
	5: // wait for request sent
		IF NOT FB_SocketSend.bBusy AND NOT FB_SocketSend.bError THEN
			ton_TimeOut.IN :=FALSE;
			FB_SocketSend.bExecute := FALSE;
			i_State := i_State+1;  
		ELSIF FB_SocketSend.bError OR ton_TimeOut.Q THEN
			FB_SocketSend.bExecute := FALSE;
			ton_TimeOut.IN :=FALSE;
			i_State := 100;
		END_IF
		
	6: // wait for data
		ton_Wait.IN := TRUE;
		IF ton_Wait.Q THEN
			FB_SocketReceive.bExecute := TRUE;
			ton_Wait.IN := FALSE;
			i_State := i_State+1; 
		END_IF		 
	
	7:	
		ton_Wait.IN := TRUE;
		IF ton_Wait.Q THEN
			ton_TimeOut.IN :=TRUE;
			i_State := i_State+1; 
		END_IF	
	
	8: // convert received data
		IF NOT FB_SocketReceive.bBusy AND NOT FB_SocketReceive.bError THEN
			int_SuccessCounter := int_SuccessCounter+1;
			ton_TimeOut.IN :=FALSE;
			FB_SocketReceive.bExecute := FALSE;
	
			FB_BYTE_TO_WORD_1(byInputValue_1 := byteReceiveString[10],byInputValue_2 := byteReceiveString[11], Ebyteorderforconvert := Ebyteorder.EBIGENDIAN, woutputvalue => );
			IF WORD_TO_LREAL(FB_BYTE_TO_WORD_1.woutputvalue) = 0 THEN
				b_MeterOnline :=FALSE;
			ELSIF WORD_TO_LREAL(FB_BYTE_TO_WORD_1.woutputvalue) = 1 THEN
				b_MeterOnline :=TRUE;
			END_IF
			
			fb_ConvertBytesToLreal(	by_InputValue_1:= byteReceiveString[12], 
									by_InputValue_2:= byteReceiveString[13], 
									by_InputValue_3:= byteReceiveString[14], 
									by_InputValue_4:= byteReceiveString[15], 
									int_Divider:= 10, 
									lreal_Output=> lreal_GridVoltage_L1_V );
									
			fb_ConvertBytesToLreal(	by_InputValue_1:= byteReceiveString[16], 
									by_InputValue_2:= byteReceiveString[17], 
									by_InputValue_3:= byteReceiveString[18], 
									by_InputValue_4:= byteReceiveString[19], 
									int_Divider:= 10, 
									lreal_Output=> lreal_GridVoltage_L2_V);
									
			fb_ConvertBytesToLreal(	by_InputValue_1:= byteReceiveString[20], 
									by_InputValue_2:= byteReceiveString[21], 
									by_InputValue_3:= byteReceiveString[22], 
									by_InputValue_4:= byteReceiveString[23], 
									int_Divider:= 10, 
									lreal_Output=> lreal_GridVoltage_L3_V);
								
			fb_ConvertBytesToLreal(	by_InputValue_1:= byteReceiveString[24], 
									by_InputValue_2:= byteReceiveString[25], 
									by_InputValue_3:= byteReceiveString[26], 
									by_InputValue_4:= byteReceiveString[27], 
									int_Divider:= 100, 
									lreal_Output=> lreal_GridCurrent_L1_A );
									
			fb_ConvertBytesToLreal(	by_InputValue_1:= byteReceiveString[24], 
									by_InputValue_2:= byteReceiveString[25], 
									by_InputValue_3:= byteReceiveString[26], 
									by_InputValue_4:= byteReceiveString[27], 
									int_Divider:= 100, 
									lreal_Output=> lreal_GridCurrent_L1_A );
									
			fb_ConvertBytesToLreal(	by_InputValue_1:= byteReceiveString[28], 
									by_InputValue_2:= byteReceiveString[29], 
									by_InputValue_3:= byteReceiveString[30], 
									by_InputValue_4:= byteReceiveString[31], 
									int_Divider:= 100, 
									lreal_Output=> lreal_GridCurrent_L2_A );
									
			fb_ConvertBytesToLreal(	by_InputValue_1:= byteReceiveString[32], 
									by_InputValue_2:= byteReceiveString[33], 
									by_InputValue_3:= byteReceiveString[34], 
									by_InputValue_4:= byteReceiveString[35], 
									int_Divider:= 100, 
									lreal_Output=> lreal_GridCurrent_L3_A );
									
			fb_ConvertBytesToLreal(	by_InputValue_1:= byteReceiveString[36], 
									by_InputValue_2:= byteReceiveString[37], 
									by_InputValue_3:= byteReceiveString[38], 
									by_InputValue_4:= byteReceiveString[39], 
									int_Divider:= 1000, 
									lreal_Output=> lreal_GridPower_kW);
									
			fb_ConvertBytesToLreal(	by_InputValue_1:= byteReceiveString[40], 
									by_InputValue_2:= byteReceiveString[41], 
									by_InputValue_3:= byteReceiveString[42], 
									by_InputValue_4:= byteReceiveString[43], 
									int_Divider:= 1000, 
									lreal_Output=> lreal_GridReactivePower_kVAr);
											
			//FB_BYTE_TO_WORD_1(byInputValue_1 := byteReceiveString[44],byInputValue_2 := byteReceiveString[45], Ebyteorderforconvert := Ebyteorder.EbigENDIAN, woutputvalue => );
			//lreal_GridPowerFactor := WORD_TO_LREAL(FB_BYTE_TO_WORD_1.woutputvalue)/1000;

			lreal_GridPowerFactor := INT_TO_LREAL(WORD_TO_INT((SHL(BYTE_TO_WORD(byteReceiveString[44]),8) + BYTE_TO_WORD(byteReceiveString[45]))))/1000;


		
			FB_BYTE_TO_WORD_1(byInputValue_1 := byteReceiveString[46],byInputValue_2 := byteReceiveString[47], Ebyteorderforconvert := Ebyteorder.EbigENDIAN, woutputvalue => );
			lreal_GridFrequency_Hz := WORD_TO_LREAL(FB_BYTE_TO_WORD_1.woutputvalue)/100;
			
			fb_ConvertBytesToLreal(	by_InputValue_1:= byteReceiveString[48], 
									by_InputValue_2:= byteReceiveString[49], 
									by_InputValue_3:= byteReceiveString[50], 
									by_InputValue_4:= byteReceiveString[51], 
									int_Divider:= 100, 
									lreal_Output=> lreal_GridEnergyDelivered_kWh);
									
			fb_ConvertBytesToLreal(	by_InputValue_1:= byteReceiveString[52], 
									by_InputValue_2:= byteReceiveString[53], 
									by_InputValue_3:= byteReceiveString[54], 
									by_InputValue_4:= byteReceiveString[55], 
									int_Divider:= 100, 
									lreal_Output=> lreal_GridEnergySupllied_kWh );
			
			fb_ConvertBytesToLreal(	by_InputValue_1:= byteReceiveString[62], 
									by_InputValue_2:= byteReceiveString[63], 
									by_InputValue_3:= byteReceiveString[64], 
									by_InputValue_4:= byteReceiveString[65], 
									int_Divider:= 10 , 
									lreal_Output=> lreal_GridVoltage_L1L2_V);

			fb_ConvertBytesToLreal(	by_InputValue_1:= byteReceiveString[66], 
									by_InputValue_2:= byteReceiveString[67], 
									by_InputValue_3:= byteReceiveString[68], 
									by_InputValue_4:= byteReceiveString[69], 
									int_Divider:= 10 , 
									lreal_Output=> lreal_GridVoltage_L2L3_V);

			fb_ConvertBytesToLreal(	by_InputValue_1:= byteReceiveString[70], 
									by_InputValue_2:= byteReceiveString[71], 
									by_InputValue_3:= byteReceiveString[72], 
									by_InputValue_4:= byteReceiveString[73], 
									int_Divider:= 10 , 
									lreal_Output=> lreal_GridVoltage_L3L1_V);

			i_State := i_State+1;
		ELSIF FB_SocketSend.bError OR ton_TimeOut.Q THEN
 			FB_SocketReceive.bExecute := FALSE;
			ton_TimeOut.IN :=FALSE;
			i_State := 100;
		END_IF
	
	9: // for for next request
		ton_WaitforNetxtRequest.IN := TRUE;
		IF NOT b_Enable THEN
			ton_WaitforNetxtRequest.IN := FALSE;
			i_State := 10;
		END_IF
		IF ton_WaitforNetxtRequest.Q THEN
			ton_WaitforNetxtRequest.IN := FALSE;
			i_State := 4;
		END_IF
		IF 	ton_ConnectionEstablised.Q THEN 
			ton_WaitforNetxtRequest.IN := FALSE;
			i_State := 10;
		END_IF

	10: // close sockets
		FB_CloseSockets.bExecute := TRUE;
		ton_TimeOut.IN :=TRUE;
		i_State := i_State+1;
		
	11: // wait for sockets closed
		
		IF NOT FB_CloseSockets.bBusy THEN
			int_ReconnectCounter := int_ReconnectCounter+1;
			FB_CloseSockets.bExecute := FALSE;
			i_State := 0;
		ELSIF FB_CloseSockets.bError THEN
			int_ReconnectCounter := int_ReconnectCounter+1;
			FB_CloseSockets.bExecute := FALSE;
			i_State := 0;
		END_IF

	100: // wait state for reconect
		
		FB_SocketConnect.bExecute := FALSE;
		FB_SocketSend.bExecute := FALSE;
		FB_SocketReceive.bExecute := FALSE;
		ton_ConnectionEstablised.IN := FALSE;
		ton_TimeOut.IN :=FALSE;
		ton_WaitforReconnect.IN := TRUE;
		IF ton_WaitforReconnect.Q THEN
			int_ErrorCount := int_ErrorCount+1;
			ton_WaitforReconnect.IN := FALSE;
			i_State := 10;
		END_IF
	
END_CASE



FB_SocketConnect(
	sSrvNetId := '',
	sRemoteHost := str_IPAdress,
	nRemotePort := 502,
	bExecute := ,
	tTimeout := T#1S,
	bBusy =>,
	bError =>,
	nErrId =>,
	hSocket => hSocket);
	
FB_SocketSend(
	sSrvNetId:= '', 
	hSocket:= hSocket, 
	cbLen:= 12,
	pSrc:= ADR( byteSendString ), 
	bExecute:= , 
	tTimeout:= T#3S, 
	bBusy=> , 
	bError=> , 
	nErrId=> );
	
FB_SocketReceive(
	sSrvNetId:= '', 
	hSocket:= hSocket, 
	cbLen:= 200, 
	pDest:= ADR( byteReceiveString ), 
	bExecute:= , 
	tTimeout:= T#3S, 
	bBusy=> , 
	bError=> , 
	nErrId=> , 
	nRecBytes=> );

FB_CloseSockets(
	sSrvNetId:= '', 
	bExecute:= , 
	tTimeout:= T#2S, 
	bBusy=> , 
	bError=> , 
	nErrId=> );
	
ton_TimeOut(PT := T#5S);
ton_WaitforReconnect(PT := T#10S);
ton_ConnectionEstablised(pt := time_ReconnectTime);
ton_WaitforNetxtRequest(PT:= T#10S);
ton_Wait(PT:=T#2S);

END_FUNCTION_BLOCK

// ---- POUs/prgGrid.TcPOU
PROGRAM prgGrid
VAR
	FB_PV1:FB_TCPModbusRequest_Grid;
	FB_PV2:FB_TCPModbusRequest_Grid;

	lreal_GridVoltage_L1L2_V_PV1		: LREAL;				//{#lynus.ag#()}
	lreal_GridVoltage_L2L3_V_PV1		: LREAL;				//{#lynus.ag#()}
	lreal_GridVoltage_L3L1_V_PV1		: LREAL;				//{#lynus.ag#()}
	lreal_GridVoltage_L1_V_PV1			: LREAL;				//{#lynus.ag#()}
	lreal_GridVoltage_L2_V_PV1			: LREAL;				//{#lynus.ag#()}
	lreal_GridVoltage_L3_V_PV1			: LREAL;				//{#lynus.ag#()}
	lreal_GridCurrent_L1_A_PV1			: LREAL;				//{#lynus.ag#()}
	lreal_GridCurrent_L2_A_PV1			: LREAL;				//{#lynus.ag#()}
	lreal_GridCurrent_L3_A_PV1			: LREAL;				//{#lynus.ag#()}
	lreal_GridPower_kW_PV1				: LREAL;				//{#lynus.ag#()}
	lreal_GridReactivePower_kVAr_PV1	: LREAL;				//{#lynus.ag#()}
	lreal_GridPowerFactor_PV1			: LREAL;				//{#lynus.ag#()}
	lreal_GridFrequency_Hz_PV1			: LREAL;				//{#lynus.ag#()}
	lreal_GridEnergyDelivered_kWh_PV1	: LREAL;				//{#lynus.ag#()}
	lreal_GridEnergySupllied_kWh_PV1	: LREAL;				//{#lynus.ag#()}
	
	lreal_GridVoltage_L1L2_V_PV2		: LREAL;				//{#lynus.ag#()}
	lreal_GridVoltage_L2L3_V_PV2		: LREAL;				//{#lynus.ag#()}
	lreal_GridVoltage_L3L1_V_PV2		: LREAL;				//{#lynus.ag#()}
	lreal_GridVoltage_L1_V_PV2			: LREAL;				//{#lynus.ag#()}
	lreal_GridVoltage_L2_V_PV2			: LREAL;				//{#lynus.ag#()}
	lreal_GridVoltage_L3_V_PV2			: LREAL;				//{#lynus.ag#()}
	lreal_GridCurrent_L1_A_PV2			: LREAL;				//{#lynus.ag#()}
	lreal_GridCurrent_L2_A_PV2			: LREAL;				//{#lynus.ag#()}
	lreal_GridCurrent_L3_A_PV2			: LREAL;				//{#lynus.ag#()}
	lreal_GridPower_kW_PV2				: LREAL;				//{#lynus.ag#()}
	lreal_GridReactivePower_kVAr_PV2	: LREAL;				//{#lynus.ag#()}
	lreal_GridPowerFactor_PV2			: LREAL;				//{#lynus.ag#()}
	lreal_GridFrequency_Hz_PV2			: LREAL;				//{#lynus.ag#()}
	lreal_GridEnergyDelivered_kWh_PV2	: LREAL;				//{#lynus.ag#()}
	lreal_GridEnergySupllied_kWh_PV2	: LREAL;				//{#lynus.ag#()}

	lreal_HousePower_kW_PV1				: LREAL;				//{#lynus.ag#()}
	lreal_HousePower_kW_PV2				: LREAL;				//{#lynus.ag#()}

END_VAR


FB_PV1	(	b_Enable:= TRUE, 
			str_IPAdress:= prgPv.FB_PV1.str_IPAdress);


FB_PV2	(	b_Enable:= TRUE, 
			str_IPAdress:= prgPv.FB_PV2.str_IPAdress);



lreal_GridVoltage_L1L2_V_PV1 	:= FB_PV1.lreal_GridVoltage_L1L2_V;
lreal_GridVoltage_L2L3_V_PV1 	:= FB_PV1.lreal_GridVoltage_L2L3_V;
lreal_GridVoltage_L3L1_V_PV1 	:= FB_PV1.lreal_GridVoltage_L3L1_V;
lreal_GridVoltage_L1_V_PV1		:= FB_PV1.lreal_GridVoltage_L1_V;
lreal_GridVoltage_L2_V_PV1		:= FB_PV1.lreal_GridVoltage_L2_V;
lreal_GridVoltage_L3_V_PV1		:= FB_PV1.lreal_GridVoltage_L3_V;
lreal_GridCurrent_L1_A_PV1		:= FB_PV1.lreal_GridCurrent_L1_A;
lreal_GridCurrent_L2_A_PV1		:= FB_PV1.lreal_GridCurrent_L2_A;
lreal_GridCurrent_L3_A_PV1		:= FB_PV1.lreal_GridCurrent_L3_A;
lreal_GridPower_kW_PV1			:= FB_PV1.lreal_GridPower_kW;
lreal_GridReactivePower_kVAr_PV1:= FB_PV1.lreal_GridReactivePower_kVAr;
lreal_GridPowerFactor_PV1		:= FB_PV1.lreal_GridPowerFactor;
lreal_GridFrequency_Hz_PV1		:= FB_PV1.lreal_GridFrequency_Hz;
lreal_GridEnergyDelivered_kWh_PV1:= FB_PV1.lreal_GridEnergyDelivered_kWh;
lreal_GridEnergySupllied_kWh_PV1 := FB_PV1.lreal_GridEnergySupllied_kWh;

lreal_HousePower_kW_PV1 := lreal_GridPower_kW_PV1 + prgPV.lrPowerPV1;

lreal_GridVoltage_L1L2_V_PV2 	:= FB_PV2.lreal_GridVoltage_L1L2_V;
lreal_GridVoltage_L2L3_V_PV2 	:= FB_PV2.lreal_GridVoltage_L2L3_V;
lreal_GridVoltage_L3L1_V_PV2 	:= FB_PV2.lreal_GridVoltage_L3L1_V;
lreal_GridVoltage_L1_V_PV2		:= FB_PV2.lreal_GridVoltage_L1_V;
lreal_GridVoltage_L2_V_PV2		:= FB_PV2.lreal_GridVoltage_L2_V;
lreal_GridVoltage_L3_V_PV2		:= FB_PV2.lreal_GridVoltage_L3_V;
lreal_GridCurrent_L1_A_PV2		:= FB_PV2.lreal_GridCurrent_L1_A;
lreal_GridCurrent_L2_A_PV2		:= FB_PV2.lreal_GridCurrent_L2_A;
lreal_GridCurrent_L3_A_PV2		:= FB_PV2.lreal_GridCurrent_L3_A;
lreal_GridPower_kW_PV2			:= FB_PV2.lreal_GridPower_kW;
lreal_GridReactivePower_kVAr_PV2:= FB_PV2.lreal_GridReactivePower_kVAr;
lreal_GridPowerFactor_PV2		:= FB_PV2.lreal_GridPowerFactor;
lreal_GridFrequency_Hz_PV2		:= FB_PV2.lreal_GridFrequency_Hz;
lreal_GridEnergyDelivered_kWh_PV2:= FB_PV2.lreal_GridEnergyDelivered_kWh;
lreal_GridEnergySupllied_kWh_PV2 := FB_PV2.lreal_GridEnergySupllied_kWh;


lreal_HousePower_kW_PV2 := lreal_GridPower_kW_PV1 + prgPV.lrPowerPV2;

END_PROGRAM
